(*pass trough*)
THIS^.pMqttPublishQueue := pMqttPublishQueue;
THIS^.MqttPublishTopicPrefix:=MQTTPublishPrefix;
THIS^.MQTTSubscribeTopicPrefix:=MQTTSubscribePrefix;
THIS^.pMqttPublishQueue:=pMqttPublishQueue;

// Dimmer specific
THIS^.OutputDimmer:=OutputDimmer;
THIS^.Qos_Dimm:=Qos_Dimm;
THIS^.Delta_Dimm:=Delta_Dimm;


SUPER^.InitBaseMqtt();
pMqttCallbackCollector^.put(instance:= THIS^); // register the FB agains the collector so mqtt events can be received
END_METHOD

METHOD InitMqttDiscovery
VAR_INPUT
	Device: POINTER TO FB_PLC_MQTT_DISCOVERY_DEVICE;
	Name: STRING(255);
	overruleId: STRING(255) := '';
	meta: STRING(255) := '';
END_VAR
VAR
	id: STRING(255);
END_VAR
IF InitMqttDone AND NOT initMqttDiscoveryDone THEN
	
	IF CommonTypesAndFunctions.StrEquals(str1:= ADR(overruleId), str2:= ADR('')) THEN
		id := CONCAT(CONCAT(THIS^.DeviceName,'_'), THIS^.InstanceNamePt^); // 'FB_DI_PB_003'
	ELSE
		id := overruleId; // 'MY_PH_GND_HALL_01'
	END_IF
	
	Device^.CreateLightDimmerEntity(
		Name := name,
		Id := Id,
		Meta := meta,
		CommandTopic := CONCAT(THIS^.MQTTSubscribeTopic,'/Q'),
		PayloadOn := 'TRUE',
		PayloadOff := 'FALSE',
		StateTopic := CONCAT(THIS^.MQTTPublishTopic,'/Q'),
		BrightnessCommandTopic := CONCAT(THIS^.MQTTSubscribeTopic,'/OUT'),
		BrightnessStateTopic := CONCAT(THIS^.MQTTPublishTopic,'/OUT'),
		BrightnessScale := 255,
		DmxChannel := THIS^.DmxChannel,
		DmxWidth := THIS^.DmxWidth,
		DmxUniverse := THIS^.DmxUniverse);

	initMqttDiscoveryDone := TRUE;
END_IF
END_METHOD

METHOD PublishReceived : BOOL
VAR_INPUT
	///Collection of recived Data
	Data: MQTT.CALLBACK_DATA;
END_VAR
//first check if Mqtt is initialized, otherwise do nothing
IF NOT(InitMqttDone) THEN
	//mark the interface call from the collector as done
	PublishReceived := TRUE;
//check if the packet is for this FB
ELSIF CONCAT(MQTTSubscribeTopic,'/Q') =  Data.TopicOut^ THEN
	IF CommonTypesAndFunctions.StrEquals(str1:= Data.PayloadString, str2:= ADR('TRUE')) THEN
		MqttHighRequest := TRUE;
	ELSIF CommonTypesAndFunctions.StrEquals(str1:= Data.PayloadString, str2:= ADR('FALSE')) THEN
		MqttLowRequest := TRUE;
	END_IF;
	
ELSIF CONCAT(MQTTSubscribeTopic,'/OUT') =  Data.TopicOut^ THEN
	IF OSCAT_BASIC.IS_CC(str:= Data.PayloadString^,cmp:='0123456789.') AND THIS^.PRIO_HIGH = FALSE THEN
		THIS^.OUT_Target:=STRING_TO_BYTE(Data.PayloadString^);
		THIS^.SoftDimToValue:=TRUE;
	END_IF
	
	
// Legacy! backwards compatiably with /+ topics instead of /#
ELSIF CommonTypesAndFunctions.StrEqualsAtStart(str1:= ADR(MQTTSubscribeTopic), str2:= Data.TopicOut) THEN
	//mark the interface call from the collector as done
	PublishReceived := TRUE;
	//now process the data
	IF CommonTypesAndFunctions.StrEquals(str1:= Data.PayloadString, str2:= ADR('TRUE')) THEN
		MqttHighRequest := TRUE;
	ELSIF CommonTypesAndFunctions.StrEquals(str1:= Data.PayloadString, str2:= ADR('FALSE')) THEN
		MqttLowRequest := TRUE;
	ELSIF OSCAT_BASIC.IS_CC(str:= Data.PayloadString^,cmp:='0123456789.') AND THIS^.PRIO_HIGH = FALSE THEN
		THIS^.OUT_Target:=STRING_TO_BYTE(Data.PayloadString^);
		THIS^.SoftDimToValue:=TRUE;
	END_IF
END_IF
END_METHOD

END_FUNCTION_BLOCK

// FB_VIRTUAL_INT_MQTT
{attribute 'reflection' := ''}
FUNCTION_BLOCK FB_VIRTUAL_INT_MQTT EXTENDS FB_MQTT_BASE IMPLEMENTS MQTT.MQTT_SUBSCRIBE_CALLBACK
VAR_INPUT
	IN: INT;
END_VAR
VAR_OUTPUT
	OUT: INT;
END_VAR
VAR
	/// Refelection: object's full instance name
	{attribute 'instance-path' := ''}
	{attribute 'noinit'}
	InstancePath: STRING;
	Startup: BOOL := TRUE;
	UpdateFlag: BOOL;
	VirtualMode: VIRTUAL_MODES;
	DefaultValue: INT;
	SetDefaultValueStartup: BOOL;
	PublishAtStartup: BOOL;
	UsePersistentAtStartup: BOOL;
	ConfirmReceival: BOOL;
	MqttMessageReceived: BOOL;
	PreviousIn: INT;
END_VAR
VAR PERSISTENT
	/// To retain output state through powercycles
	PreviousState: INT;
END_VAR

IF VirtualMode = VIRTUAL_MODES.Output THEN
	IF (Startup AND PublishAtStartup) OR (UpdateFlag OR IN <> PreviousIn) AND InitMqttDone THEN
	pMqttPublishQueue^.AddMessage(
		Payload := INT_TO_STRING(IN),
		Topic := CONCAT(MqttPublishTopicPrefix^, MqttPublishTopicSuffix),
		Qos := MqttQos,
		MqttRetain := MqttRetain
	);
	Startup:=FALSE;
	UpdateFlag := FALSE;
	PreviousIn := IN;
	END_IF
ELSIF VirtualMode = VIRTUAL_MODES.Input THEN
	IF Startup AND SetDefaultValueStartup THEN
		OUT := DefaultValue;
	ELSIF UsePersistentAtStartup THEN
		OUT := PreviousState;
	END_IF	
	
	IF ((Startup AND PublishAtStartup) OR (ConfirmReceival AND MqttMessageReceived)) AND InitMqttDone THEN
	pMqttPublishQueue^.AddMessage(
		Payload := INT_TO_STRING(OUT),
		Topic := CONCAT(MqttPublishTopicPrefix^, MqttPublishTopicSuffix),
		Qos := MqttQos,
		MqttRetain := MqttRetain
	);
	Startup:=FALSE;
	MqttMessageReceived := FALSE;
	PreviousState:=OUT;
	END_IF		
	
END_IF

METHOD ConfigureFunctionBlockAsVirtualInput : BOOL
VAR_INPUT
	DefaultValue: INT;
	SetDefaultValueStartup: BOOL;
	PublishAtStartup: BOOL;
	UsePersistentAtStartup: BOOL;
	ConfirmReceival: BOOL;
END_VAR
THIS^.DefaultValue:=DefaultValue;
THIS^.SetDefaultValueStartup:=SetDefaultValueStartup;
THIS^.PublishAtStartup:=PublishAtStartup;
THIS^.UsePersistentAtStartup:=UsePersistentAtStartup;
THIS^.ConfirmReceival:=ConfirmReceival;
THIS^.VirtualMode:=VIRTUAL_MODES.Input;
END_METHOD

METHOD ConfigureFunctionBlockAsVirtualOutput : BOOL
VAR_INPUT
	PublishAtStartup: BOOL;
END_VAR
THIS^.PublishAtStartup:=PublishAtStartup;
THIS^.VirtualMode:=VIRTUAL_MODES.Output;
END_METHOD

METHOD InitMqtt
VAR_INPUT
	MQTTPublishPrefix: POINTER TO STRING;
	MQTTSubscribePrefix: POINTER TO STRING;
	pMqttPublishQueue: POINTER TO FB_MqttPublishQueue;
	pMqttCallbackCollector: POINTER TO MQTT.CallbackCollector;
	MqttQos: MQTT.QoS;
	MqttRetain: BOOL;
END_VAR
InitMqttDone := TRUE;

SUPER^._InstancePath := THIS^.InstancePath; // Due to reflection its location is important

(*pass trough*)
THIS^.pMqttPublishQueue := pMqttPublishQueue;
THIS^.MqttPublishTopicPrefix:=MQTTPublishPrefix;
THIS^.MQTTSubscribeTopicPrefix:=MQTTSubscribePrefix;
THIS^.pMqttPublishQueue:=pMqttPublishQueue;
THIS^.MqttQos:=MqttQos;
THIS^.MqttRetain:=MqttRetain;


SUPER^.InitBaseMqtt();
pMqttCallbackCollector^.put(instance:= THIS^); // register the FB agains the collector so mqtt events can be received
END_METHOD

METHOD PublishReceived : BOOL
VAR_INPUT
	///Collection of recived Data
	Data: MQTT.CALLBACK_DATA;
END_VAR
//first check if Mqtt is initialized and FB in input mode, otherwise do nothing
IF NOT(InitMqttDone) AND VirtualMode <> VIRTUAL_MODES.Input THEN
	//mark the interface call from the collector as done
	PublishReceived := TRUE;
//check if the packet is for this FB
ELSIF CommonTypesAndFunctions.StrEquals(str1:= ADR(MQTTSubscribeTopic), str2:= Data.TopicOut) THEN
	//mark the interface call from the collector as done
	PublishReceived := TRUE;
	//process the data
	IF OSCAT_BASIC.IS_NUM(str:= Data.PayloadString^) THEN
		THIS^.OUT := STRING_TO_INT(Data.PayloadString^);	
		MqttMessageReceived := TRUE;	
	END_IF
END_IF
END_METHOD

METHOD SetValue : BOOL
VAR_INPUT
	Value: INT;
END_VAR
THIS^.OUT:=Value;
THIS^.UpdateFlag:=TRUE;
END_METHOD

END_FUNCTION_BLOCK

// FB_VIRTUAL_BOOL_MQTT
{attribute 'reflection' := ''}
FUNCTION_BLOCK FB_VIRTUAL_BOOL_MQTT EXTENDS FB_MQTT_BASE IMPLEMENTS MQTT.MQTT_SUBSCRIBE_CALLBACK
VAR_INPUT
	IN: BOOL;
END_VAR
VAR_OUTPUT
	OUT: BOOL;
END_VAR
VAR
	/// Refelection: object's full instance name
	{attribute 'instance-path' := ''}
	{attribute 'noinit'}
	InstancePath: STRING;
	Startup: BOOL := TRUE;
	UpdateFlag: BOOL;
	VirtualMode: VIRTUAL_MODES;
	DefaultValue: BOOL;
	SetDefaultValueStartup: BOOL;
	PublishAtStartup: BOOL;
	UsePersistentAtStartup: BOOL;
	ConfirmReceival: BOOL;
	MqttMessageReceived: BOOL;
	PreviousIn: BOOL;
END_VAR
VAR PERSISTENT
	/// To retain output state through powercycles
	PreviousState: BOOL;
END_VAR

IF VirtualMode = VIRTUAL_MODES.Output THEN
	IF (Startup AND PublishAtStartup) OR (UpdateFlag OR IN <> PreviousIn) AND InitMqttDone THEN
	pMqttPublishQueue^.AddMessage(
		Payload := BOOL_TO_STRING(IN),
		Topic := CONCAT(MqttPublishTopicPrefix^, MqttPublishTopicSuffix),
		Qos := MqttQos,
		MqttRetain := MqttRetain
	);
	Startup:=FALSE;
	UpdateFlag := FALSE;
	PreviousIn := IN;
	END_IF
ELSIF VirtualMode = VIRTUAL_MODES.Input THEN
	IF Startup AND SetDefaultValueStartup THEN
		OUT := DefaultValue;
	ELSIF UsePersistentAtStartup THEN
		OUT := PreviousState;
	END_IF	
	
	IF ((Startup AND PublishAtStartup) OR (ConfirmReceival AND MqttMessageReceived)) AND InitMqttDone THEN
	pMqttPublishQueue^.AddMessage(
		Payload := BOOL_TO_STRING(OUT),
		Topic := CONCAT(MqttPublishTopicPrefix^, MqttPublishTopicSuffix),
		Qos := MqttQos,
		MqttRetain := MqttRetain
	);
	Startup:=FALSE;
	MqttMessageReceived := FALSE;
	PreviousState:=OUT;
	END_IF		
	
END_IF

METHOD ConfigureFunctionBlockAsVirtualInput : BOOL
VAR_INPUT
	DefaultValue: BOOL;
	SetDefaultValueStartup: BOOL;
	PublishAtStartup: BOOL;
	UsePersistentAtStartup: BOOL;
	ConfirmReceival: BOOL;
END_VAR
THIS^.DefaultValue:=DefaultValue;
THIS^.SetDefaultValueStartup:=SetDefaultValueStartup;
THIS^.PublishAtStartup:=PublishAtStartup;
THIS^.UsePersistentAtStartup:=UsePersistentAtStartup;
THIS^.ConfirmReceival:=ConfirmReceival;
THIS^.VirtualMode:=VIRTUAL_MODES.Input;
END_METHOD

METHOD ConfigureFunctionBlockAsVirtualOutput : BOOL
VAR_INPUT
	PublishAtStartup: BOOL;
END_VAR
THIS^.PublishAtStartup:=PublishAtStartup;
THIS^.VirtualMode:=VIRTUAL_MODES.Output;
END_METHOD

METHOD InitMqtt
VAR_INPUT
	MQTTPublishPrefix: POINTER TO STRING;
	MQTTSubscribePrefix: POINTER TO STRING;
	pMqttPublishQueue: POINTER TO FB_MqttPublishQueue;
	pMqttCallbackCollector: POINTER TO MQTT.CallbackCollector;
	MqttQos: MQTT.QoS;
	MqttRetain: BOOL;
END_VAR
InitMqttDone := TRUE;

SUPER^._InstancePath := THIS^.InstancePath; // Due to reflection its location is important

(*pass trough*)
THIS^.pMqttPublishQueue := pMqttPublishQueue;
THIS^.MqttPublishTopicPrefix:=MQTTPublishPrefix;
THIS^.MQTTSubscribeTopicPrefix:=MQTTSubscribePrefix;
THIS^.pMqttPublishQueue:=pMqttPublishQueue;
THIS^.MqttQos:=MqttQos;
THIS^.MqttRetain:=MqttRetain;


SUPER^.InitBaseMqtt();
pMqttCallbackCollector^.put(instance:= THIS^); // register the FB agains the collector so mqtt events can be received
END_METHOD

METHOD PublishReceived : BOOL
VAR_INPUT
	///Collection of recived Data
	Data: MQTT.CALLBACK_DATA;
END_VAR
//first check if Mqtt is initialized and FB in input mode, otherwise do nothing
IF NOT(InitMqttDone) AND VirtualMode <> VIRTUAL_MODES.Input THEN
	//mark the interface call from the collector as done
	PublishReceived := TRUE;
//check if the packet is for this FB
ELSIF CommonTypesAndFunctions.StrEquals(str1:= ADR(MQTTSubscribeTopic), str2:= Data.TopicOut) THEN
	//mark the interface call from the collector as done
	PublishReceived := TRUE;
	//process the data
	IF CommonTypesAndFunctions.StrEquals(str1:= Data.PayloadString, str2:= ADR('TRUE')) THEN
		THIS^.OUT := TRUE;
		MqttMessageReceived := TRUE;
	END_IF
	IF CommonTypesAndFunctions.StrEquals(str1:= Data.PayloadString, str2:= ADR('FALSE')) THEN
		THIS^.OUT := FALSE;
		MqttMessageReceived := TRUE;
	END_IF
END_IF
END_METHOD

METHOD SetValue : BOOL
VAR_INPUT
	Value: BOOL;
END_VAR
THIS^.OUT:=Value;
THIS^.UpdateFlag:=TRUE;
END_METHOD

END_FUNCTION_BLOCK

// FB_VIRTUAL_STRING_MQTT
{attribute 'reflection' := ''}
FUNCTION_BLOCK FB_VIRTUAL_STRING_MQTT EXTENDS FB_MQTT_BASE IMPLEMENTS MQTT.MQTT_SUBSCRIBE_CALLBACK
VAR_INPUT
	IN: STRING;
END_VAR
VAR_OUTPUT
	OUT: STRING;
END_VAR
VAR
	/// Refelection: object's full instance name
	{attribute 'noinit'}
	{attribute 'instance-path' := ''}
	InstancePath: STRING;
	Startup: BOOL := TRUE;
	UpdateFlag: BOOL;
	VirtualMode: VIRTUAL_MODES;
	DefaultValue: STRING;
	SetDefaultValueStartup: BOOL;
	PublishAtStartup: BOOL;
	UsePersistentAtStartup: BOOL;
	ConfirmReceival: BOOL;
	MqttMessageReceived: BOOL;
	PreviousIn: STRING;
END_VAR
VAR PERSISTENT
	/// To retain output state through powercycles
	PreviousState: STRING;
END_VAR

IF VirtualMode = VIRTUAL_MODES.Output THEN
	IF (Startup AND PublishAtStartup) OR (UpdateFlag OR IN <> PreviousIn) AND InitMqttDone THEN
	pMqttPublishQueue^.AddMessage(
		Payload := IN,
		Topic := CONCAT(MqttPublishTopicPrefix^, MqttPublishTopicSuffix),
		Qos := MqttQos,
		MqttRetain := MqttRetain
	);
	Startup:=FALSE;
	UpdateFlag := FALSE;
	PreviousIn := IN;
	END_IF
ELSIF VirtualMode = VIRTUAL_MODES.Input THEN
	IF Startup AND SetDefaultValueStartup THEN
		OUT := DefaultValue;
	ELSIF UsePersistentAtStartup THEN
		OUT := PreviousState;
	END_IF	
	
	IF ((Startup AND PublishAtStartup) OR (ConfirmReceival AND MqttMessageReceived)) AND InitMqttDone THEN
	pMqttPublishQueue^.AddMessage(
		Payload := OUT,
		Topic := CONCAT(MqttPublishTopicPrefix^, MqttPublishTopicSuffix),
		Qos := MqttQos,
		MqttRetain := MqttRetain
	);
	Startup:=FALSE;
	MqttMessageReceived := FALSE;
	PreviousState:=OUT;
	END_IF		
	
END_IF

METHOD ConfigureFunctionBlockAsVirtualInput : BOOL
VAR_INPUT
	DefaultValue: STRING;
	SetDefaultValueStartup: BOOL;
	PublishAtStartup: BOOL;
	UsePersistentAtStartup: BOOL;
	ConfirmReceival: BOOL;
END_VAR
THIS^.DefaultValue:=DefaultValue;
THIS^.SetDefaultValueStartup:=SetDefaultValueStartup;
THIS^.PublishAtStartup:=PublishAtStartup;
THIS^.UsePersistentAtStartup:=UsePersistentAtStartup;
THIS^.ConfirmReceival:=ConfirmReceival;
THIS^.VirtualMode:=VIRTUAL_MODES.Input;
END_METHOD

METHOD ConfigureFunctionBlockAsVirtualOutput : BOOL
VAR_INPUT
	PublishAtStartup: BOOL;
END_VAR
THIS^.PublishAtStartup:=PublishAtStartup;
THIS^.VirtualMode:=VIRTUAL_MODES.Output;
END_METHOD

METHOD InitMqtt
VAR_INPUT
	MQTTPublishPrefix: POINTER TO STRING;
	MQTTSubscribePrefix: POINTER TO STRING;
	pMqttPublishQueue: POINTER TO FB_MqttPublishQueue;
	pMqttCallbackCollector: POINTER TO MQTT.CallbackCollector;
	MqttQos: MQTT.QoS;
	MqttRetain: BOOL;
END_VAR
InitMqttDone := TRUE;

SUPER^._InstancePath := THIS^.InstancePath; // Due to reflection its location is important

(*pass trough*)
THIS^.pMqttPublishQueue := pMqttPublishQueue;
THIS^.MqttPublishTopicPrefix:=MQTTPublishPrefix;
THIS^.MQTTSubscribeTopicPrefix:=MQTTSubscribePrefix;
THIS^.pMqttPublishQueue:=pMqttPublishQueue;
THIS^.MqttQos:=MqttQos;
THIS^.MqttRetain:=MqttRetain;


SUPER^.InitBaseMqtt();
pMqttCallbackCollector^.put(instance:= THIS^); // register the FB agains the collector so mqtt events can be received
END_METHOD

METHOD PublishReceived : BOOL
VAR_INPUT
	///Collection of recived Data
	Data: MQTT.CALLBACK_DATA;
END_VAR
//first check if Mqtt is initialized and FB in input mode, otherwise do nothing
IF NOT(InitMqttDone) AND VirtualMode <> VIRTUAL_MODES.Input THEN
	//mark the interface call from the collector as done
	PublishReceived := TRUE;
//check if the packet is for this FB
ELSIF CommonTypesAndFunctions.StrEquals(str1:= ADR(MQTTSubscribeTopic), str2:= Data.TopicOut) THEN
	//mark the interface call from the collector as done
	PublishReceived := TRUE;
	//process the data
	THIS^.OUT := Data.PayloadString^;	
	MqttMessageReceived := TRUE;
END_IF
END_METHOD

METHOD SetValue : BOOL
VAR_INPUT
	Value: STRING;
END_VAR
THIS^.OUT:=Value;
THIS^.UpdateFlag:=TRUE;
END_METHOD

END_FUNCTION_BLOCK

// FB_VIRTUAL_REAL_MQTT
{attribute 'reflection' := ''}
FUNCTION_BLOCK FB_VIRTUAL_REAL_MQTT EXTENDS FB_MQTT_BASE IMPLEMENTS MQTT.MQTT_SUBSCRIBE_CALLBACK
VAR_INPUT
	IN: REAL;
END_VAR
VAR_OUTPUT
	OUT: REAL;
END_VAR
VAR
	/// Refelection: object's full instance name
	{attribute 'instance-path' := ''}
	{attribute 'noinit'}
	InstancePath: STRING;
	Startup: BOOL := TRUE;
	UpdateFlag: BOOL;
	VirtualMode: VIRTUAL_MODES;
	DefaultValue: REAL;
	SetDefaultValueStartup: BOOL;
	PublishAtStartup: BOOL;
	UsePersistentAtStartup: BOOL;
	ConfirmReceival: BOOL;
	MqttMessageReceived: BOOL;
	PreviousIn: REAL;
END_VAR
VAR PERSISTENT
	/// To retain output state through powercycles
	PreviousState: REAL;
END_VAR

IF VirtualMode = VIRTUAL_MODES.Output THEN
	IF (Startup AND PublishAtStartup) OR (UpdateFlag OR IN <> PreviousIn) AND InitMqttDone THEN
	pMqttPublishQueue^.AddMessage(
		Payload := REAL_TO_STRING(IN),
		Topic := CONCAT(MqttPublishTopicPrefix^, MqttPublishTopicSuffix),
		Qos := MqttQos,
		MqttRetain := MqttRetain
	);
	Startup:=FALSE;
	UpdateFlag := FALSE;
	PreviousIn := IN;
	END_IF
ELSIF VirtualMode = VIRTUAL_MODES.Input THEN
	IF Startup AND SetDefaultValueStartup THEN
		OUT := DefaultValue;
	ELSIF UsePersistentAtStartup THEN
		OUT := PreviousState;
	END_IF	
	
	IF ((Startup AND PublishAtStartup) OR (ConfirmReceival AND MqttMessageReceived)) AND InitMqttDone THEN
	pMqttPublishQueue^.AddMessage(
		Payload := REAL_TO_STRING(OUT),
		Topic := CONCAT(MqttPublishTopicPrefix^, MqttPublishTopicSuffix),
		Qos := MqttQos,
		MqttRetain := MqttRetain
	);
	Startup:=FALSE;
	MqttMessageReceived := FALSE;
	PreviousState:=OUT;
	END_IF		
	
END_IF

METHOD ConfigureFunctionBlockAsVirtualInput : BOOL
VAR_INPUT
	DefaultValue: REAL;
	SetDefaultValueStartup: BOOL;
	PublishAtStartup: BOOL;
	UsePersistentAtStartup: BOOL;
	ConfirmReceival: BOOL;
END_VAR
THIS^.DefaultValue:=DefaultValue;
THIS^.SetDefaultValueStartup:=SetDefaultValueStartup;
THIS^.PublishAtStartup:=PublishAtStartup;
THIS^.UsePersistentAtStartup:=UsePersistentAtStartup;
THIS^.ConfirmReceival:=ConfirmReceival;
THIS^.VirtualMode:=VIRTUAL_MODES.Input;
END_METHOD

METHOD ConfigureFunctionBlockAsVirtualOutput : BOOL
VAR_INPUT
	PublishAtStartup: BOOL;
END_VAR
THIS^.PublishAtStartup:=PublishAtStartup;
THIS^.VirtualMode:=VIRTUAL_MODES.Output;
END_METHOD

METHOD InitMqtt
VAR_INPUT
	MQTTPublishPrefix: POINTER TO STRING;
	MQTTSubscribePrefix: POINTER TO STRING;
	pMqttPublishQueue: POINTER TO FB_MqttPublishQueue;
	pMqttCallbackCollector: POINTER TO MQTT.CallbackCollector;
	MqttQos: MQTT.QoS;
	MqttRetain: BOOL;
END_VAR
InitMqttDone := TRUE;

SUPER^._InstancePath := THIS^.InstancePath; // Due to reflection its location is important

(*pass trough*)
THIS^.pMqttPublishQueue := pMqttPublishQueue;
THIS^.MqttPublishTopicPrefix:=MQTTPublishPrefix;
THIS^.MQTTSubscribeTopicPrefix:=MQTTSubscribePrefix;
THIS^.pMqttPublishQueue:=pMqttPublishQueue;
THIS^.MqttQos:=MqttQos;
THIS^.MqttRetain:=MqttRetain;


SUPER^.InitBaseMqtt();
pMqttCallbackCollector^.put(instance:= THIS^); // register the FB agains the collector so mqtt events can be received
END_METHOD

METHOD PublishReceived : BOOL
VAR_INPUT
	///Collection of recived Data
	Data: MQTT.CALLBACK_DATA;
END_VAR
//first check if Mqtt is initialized and FB in input mode, otherwise do nothing
IF NOT(InitMqttDone) AND VirtualMode <> VIRTUAL_MODES.Input THEN
	//mark the interface call from the collector as done
	PublishReceived := TRUE;
//check if the packet is for this FB
ELSIF CommonTypesAndFunctions.StrEquals(str1:= ADR(MQTTSubscribeTopic), str2:= Data.TopicOut) THEN
	//mark the interface call from the collector as done
	PublishReceived := TRUE;
	//process the data
	THIS^.OUT := STRING_TO_REAL(Data.PayloadString^);	
	MqttMessageReceived := TRUE;	
END_IF
END_METHOD

METHOD SetValue : BOOL
VAR_INPUT
	Value: REAL;
END_VAR
THIS^.OUT:=Value;
THIS^.UpdateFlag:=TRUE;
END_METHOD

END_FUNCTION_BLOCK

// HomeAutomation/PRG's/PLC_PRG_MQTT
PROGRAM PLC_PRG_MQTT
VAR
	MQTTClient				:MQTT.MQTTClient;
	MQTT_IN_OUT				:MQTT.MQTT_IN_OUT;
	MQTTInfo				:MQTT.MQTT_INFO;
	MQTTBirthMessage		:MQTT_MESSAGE;;
	MQTTBirthHartbeat		:OSCAT_BASIC.GEN_PULSE;
	MQTTConnectTrigger		:Standard.R_TRIG;
	MQTTPublishBirth		:BOOL:=TRUE;
	MQTTBirthPublisher		:FB_MqttPublishWorker;

	(* variables for MQTT setup *)
	initMqtt				:BOOL;
	icounter				:UDINT;
	
	(* variables for MQTT publishing *)
	ipublishers				:UDINT:=40;
	publishers				:ARRAY[0..39] OF FB_MqttPublishWorker;
	
	(* variables to work with Mqttbuffer *)
	i : UDINT;
	
	(* variables for MQTT subscribing *)
	subscriber_FB_OUTPUT_SWITCH_MQTT:MQTT.MQTTSubscribe;
	subscriber_FB_OUTPUT_COVER_MQTT:MQTT.MQTTSubscribe;	
	subscriber_FB_VIRTUAL_MQTT:MQTT.MQTTSubscribe;	
	subscriber_FB_DIMMER_MQTT:MQTT.MQTTSubscribe;
	subscriber_FB_RS485_MQTT:MQTT.MQTTSubscribe;	
END_VAR

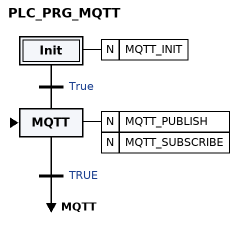
INITIAL_STEP Init:
    MQTT_INIT(N);
END_STEP
TRANSITION FROM Init TO MQTT
    := True;
END_TRANSITION
STEP MQTT:
    MQTT_PUBLISH(N);
    MQTT_SUBSCRIBE(N);
END_STEP
TRANSITION FROM MQTT TO MQTT
    := TRUE;
END_TRANSITION

ACTION MQTT_INIT:

IF NOT initMqtt THEN
	initMqtt := TRUE;
	(* Basic MQTT config *)
	MQTT_IN_OUT.ClientID := MqttVariables.clientID;
	
	(* Set the LWT topic / payload *)
	MQTT_IN_OUT.BuildWillTopicAndMessage := FALSE;
	MQTT_IN_OUT.WillTopicBase := '';
	MQTT_IN_OUT.ClientWillTopic := MqttVariables.MqttAvailabilityTopic;
	MQTT_IN_OUT.ClientWillMessage := MqttVariables.MqttAvailabilityOfflinePayload;
	
	(* Set the birth message *)
	MQTTBirthMessage.Payload := MqttVariables.MqttAvailabilityOnlinePayload;
	MQTTBirthMessage.Topic := MqttVariables.MqttAvailabilityTopic;
	MQTTBirthMessage.Qos := MqttVariables.MQTT_QOS_EXACTLY_ONCE;
	MQTTBirthMessage.MqttRetain := FALSE;
	
	(* Configure the rising edge detector to detect a connect/reconnect to the broker, used for  birth message *)
	MQTTConnectTrigger(CLK := MQTTInfo.MQTT_CONNECTED);
	
	(* Configure the dedicated MQTTBirth publisher *)
	MQTTBirthPublisher.Init(inputMQTT_IN_OUT:= ADR(MQTT_IN_OUT));
	
	(* Configure the pulse generator for the birth message hartbeat *)
	 MQTTBirthHartbeat(ENQ:=TRUE, PTH:=T#0S, PTL:=MqttVariables.MQTTAvailabilityHartbeatTime);
	
	(* INIT MQTT PUBLISH STUFF *)
	FOR icounter := 0 TO (ipublishers-1) DO		
		publishers[icounter].Init(inputMQTT_IN_OUT:= ADR(MQTT_IN_OUT));
	END_FOR 
	
	(* INIT MQTT SUBSCRIBE STUFF *)
	subscriber_FB_OUTPUT_SWITCH_MQTT.SetMqttInOut(MQTT_IN_OUT:= MQTT_IN_OUT);	
	subscriber_FB_OUTPUT_COVER_MQTT.SetMqttInOut(MQTT_IN_OUT:= MQTT_IN_OUT);
	subscriber_FB_VIRTUAL_MQTT.SetMqttInOut(MQTT_IN_OUT:= MQTT_IN_OUT);	
	subscriber_FB_DIMMER_MQTT.SetMqttInOut(MQTT_IN_OUT:= MQTT_IN_OUT);
	subscriber_FB_RS485_MQTT.SetMqttInOut(MQTT_IN_OUT:= MQTT_IN_OUT);
END_IF
END_ACTION

ACTION MQTT_PUBLISH:
(* set user led green if connected to MQTT broker, flashing red if not *)
(* é!COCKPIT version *)
(* LED_1_BrokerStatus(eID:=eLedID.AppLED_1, xOpen:=TRUE );
IF(MQTTClient.connected) THEN
	LED_1_BrokerStatus.SetStatic(eLedColor.Green);
ELSE
	LED_1_BrokerStatus.SetFlash(T#1S,eLedColor.Red, eLedColor.Off);  
END_IF *)
(* Codesys 3S version *)
(*
IF MQTTClient.connected THEN
     PFC.SetLed(which:=PFC.LED.U1, how:=PFC.LedState.STATIC_GRN);
ELSE
     PFC.SetLed(which:=PFC.LED.U1, how:=PFC.LedState.BLINK_RED);
END_IF 
*)

(* allow the rising edge detector to detect a connect/reconnect to the broker, used for  birth message *)
MQTTConnectTrigger(CLK := MQTTInfo.MQTT_CONNECTED);

(* allow the pulse generator to generate a pulse, used for birth message hartbeat *)
MQTTBirthHartbeat(ENQ:=TRUE, PTH:=T#0S, PTL:=MqttVariables.MQTTAvailabilityHartbeatTime);

(* Check if this is a new connection due to startup or connection issues *)
IF initMqtt AND (MQTTConnectTrigger.Q OR MQTTBirthHartbeat.Q) THEN
	MQTTPublishBirth := TRUE;
END_IF

(* On connect or reconnect publish a birth message using the dedicated birth publisher *)
IF MQTTPublishBirth THEN
	MQTTBirthPublisher.PublishMessage(MqttMessage := MQTTBirthMessage);
	MQTTPublishBirth:=FALSE;
END_IF


(* Check if Mqtt is initialized AND if there are elements on the queue to process AND if a MQTTbirthmessage has been published successfully *)
IF initMqtt AND NOT(MqttVariables.fbMqttPublishQueue.EMPTY) AND MQTTPublishBirth = FALSE AND MQTTBirthPublisher.SendDone THEN	
	(* Loop through all free publishers untill there are no more elements in the queue or no more free publishers *)
	FOR i:=0 TO (ipublishers-1) DO			
		(* use the publishers that are free  *)
		IF publishers[i].SendDone AND NOT(MqttVariables.fbMqttPublishQueue.EMPTY) THEN	
			(* Pass message from the queue to a publisher *)
			publishers[i].PublishMessage(MqttMessage:= MqttVariables.fbMqttPublishQueue.GetMessage());
		ELSIF MqttVariables.fbMqttPublishQueue.EMPTY THEN
			(* Queue is empty, jump out of the for loop	*)
			EXIT;	
		END_IF
	END_FOR
END_IF


(* If MQTT is initialized, let the MqttPublishWorkers do their work *)
IF initMqtt THEN	
	MQTT_IN_OUT.clientFB(
		MQTT_IN_OUT:= MQTT_IN_OUT, 
		ENABLE:= TRUE, 
		URL:= MQttVariables.broker, 
		TIMEOUT:= T#1S, 
		TLS:= FALSE);		
		
	MQTTBirthPublisher();
	
	FOR i := 0 TO (ipublishers-1) DO
  		publishers[i]();
	END_FOR

END_IF
END_ACTION

ACTION MQTT_SUBSCRIBE:
(* If MQTT is initialized, let the subscriber(s) do its work *)
IF initMqtt THEN
	
	MQTT_IN_OUT.clientFB(
		MQTT_IN_OUT:= MQTT_IN_OUT, 
		ENABLE:= TRUE, 
		URL:= MqttVariables.broker, 
		TIMEOUT:= T#1S, 
		TLS:= FALSE);

	subscriber_FB_OUTPUT_SWITCH_MQTT(
		Subscribe:= TRUE, 
		Topic:= ADR(MqttVariables.MqttSubSwitchTopic), 
		QoSSubscribe:= MqttVariables.MQTT_QOS_EXACTLY_ONCE, 
		ExpectingString:= TRUE, 
		Callback:= MqttVariables.collector_FB_OUTPUT_SWITCH_MQTT,
	);	
	subscriber_FB_OUTPUT_COVER_MQTT(
		Subscribe:= TRUE, 
		Topic:= ADR(MqttVariables.MqttSubCoverTopic), 
		QoSSubscribe:= MqttVariables.MQTT_QOS_EXACTLY_ONCE, 
		ExpectingString:= TRUE, 
		Callback:= MqttVariables.collector_FB_OUTPUT_COVER_MQTT,
	);	
	subscriber_FB_VIRTUAL_MQTT(
		Subscribe:= TRUE, 
		Topic:= ADR(MqttVariables.MqttSubVirtualTopic), 
		QoSSubscribe:= MqttVariables.MQTT_QOS_EXACTLY_ONCE, 
		ExpectingString:= TRUE, 
		Callback:= MqttVariables.collector_FB_VIRTUAL_MQTT,
	);
	subscriber_FB_DIMMER_MQTT(
		Subscribe:= TRUE, 
		Topic:= ADR(MqttVariables.MqttSubDimmerTopic), 
		QoSSubscribe:= MqttVariables.MQTT_QOS_EXACTLY_ONCE, 
		ExpectingString:= TRUE, 
		Callback:= MqttVariables.collector_FB_DIMMER_MQTT,
	);
	subscriber_FB_RS485_MQTT(
		Subscribe:= TRUE, 
		Topic:= ADR(MqttVariables.MqttSubRS485Topic), 
		QoSSubscribe:= MqttVariables.MQTT_QOS_EXACTLY_ONCE,
		ExpectingString:= TRUE, 
		Callback:= MqttVariables.collector_FB_RS485_MQTT,
	);
END_IF
END_ACTION

END_PROGRAM

// Mqtt/FB_MqttPublishWorker
FUNCTION_BLOCK FB_MqttPublishWorker
VAR_OUTPUT
	SendDone: BOOL;
END_VAR
VAR
	LocalMqttMessage: MQTT_MESSAGE;
	InitDone: BOOL;
	RequestToSend: BOOL;
	Send: BOOL;
	publish: MQTT.MQTTPublish;
END_VAR

//need to call publish here because of FB nums
publish(
	Topic:= ADR(LocalMqttMessage.Topic), 
	PayloadString:= ADR(LocalMqttMessage.Payload), 
	PublishAsString:= TRUE, 
	QoSIn:= LocalMqttMessage.Qos, 
	MRetain:= LocalMqttMessage.MqttRetain, 
	send:= Send);
	
IF NOT InitDone THEN RETURN; END_IF

IF RequestToSend THEN
	Send := TRUE;
	SendDone := FALSE;
END_IF

IF publish.done THEN
	 SendDone := TRUE;
	 RequestToSend:=FALSE;
	 Send:=FALSE;
END_IF

METHOD Init
VAR_INPUT
	///Pointer MQTTT exchange strucure
	inputMQTT_IN_OUT: POINTER TO MQTT.MQTT_IN_OUT;
END_VAR
publish.SetMqttInOut(MQTT_IN_OUT := inputMQTT_IN_OUT^);

InitDone := TRUE;
SendDone := TRUE;
END_METHOD

METHOD PublishMessage
VAR_INPUT
	MqttMessage: MQTT_MESSAGE;
END_VAR
LocalMqttMessage := MqttMessage;

RequestToSend:=TRUE;
END_METHOD

END_FUNCTION_BLOCK

// HomeAutomation/PRG's/DMX_SEND
PROGRAM DMX_SEND
VAR
	Universe	: INT     :=1;
	IP_CONTROL2	: oscat_network.IP_CONTROL2;
	IP_C		: oscat_network.IP_C;
	S_BUF1		: oscat_network.NETWORK_BUFFER_SHORT;
	R_BUF1		: oscat_network.NETWORK_BUFFER_SHORT;
	error_send	: BOOL:= FALSE;
	i			: INT;
	init		: BOOL;
	start		: INT;
	size		: INT;
	LED_1_BrokerStatus		:FbAppLED;
	Step: INT:=0;
END_VAR

IF init = FALSE THEN
	init := TRUE;
	//https://art-net.org.uk/how-it-works/streaming-packets/artdmx-packet-definition/
	(* Write DMX header character in the buffer *) 
	S_BUF1.BUFFER [0]:= BYTE#16#41; // A
	S_BUF1.BUFFER [1]:= BYTE#16#72; // R	
	S_BUF1.BUFFER [2]:= BYTE#16#74; // T
	S_BUF1.BUFFER [3]:= BYTE#16#2D; // -
	S_BUF1.BUFFER [4]:= BYTE#16#4E; // N
	S_BUF1.BUFFER [5]:= BYTE#16#65; // E
	S_BUF1.BUFFER [6]:= BYTE#16#74; // T
	S_BUF1.BUFFER [7]:= BYTE#16#00; // 0 zero
	
	S_BUF1.BUFFER [8]:= BYTE#16#00;	// Opcode ArtDMX (0x5000) little endian
	S_BUF1.BUFFER [9]:= BYTE#16#50; // Opcode ArtDMX (0x5000) little endian
	
	S_BUF1.BUFFER [10]:= BYTE#16#00; // Protocol Version Hi (0)
	S_BUF1.BUFFER [11]:= BYTE#16#0E; // Protocol Version Lo (14)
	
	S_BUF1.BUFFER [12]:= BYTE#16#00; // Sequence
	S_BUF1.BUFFER [13]:= BYTE#16#00; // Physical
	
	S_BUF1.BUFFER [16]:= BYTE#16#02; // Length Hi
	S_BUF1.BUFFER [17]:= BYTE#16#00; // Length Lo (2 to 512, even)
	(* the DMX channels that are next have already been written to the buffer *) 
	
	IF Universe = 1 THEN
		S_BUF1.BUFFER [14]:= BYTE#16#01; // Universe little endian
		S_BUF1.BUFFER [15]:= BYTE#16#00; // Universe little endian
	END_IF
	IF Universe = 2 THEN
		S_BUF1.BUFFER [14]:= BYTE#16#02; // Universe little endian
		S_BUF1.BUFFER [15]:= BYTE#16#00; // Universe little endian
	END_IF
END_IF;


size := 512+18;
FOR i:= 0 TO size DO (* check whether the DMX values ​​in the global variable have changed *)
	// i+2 is strange, buffers are not the same, its often offset with 2 sometimes by 1, todo
	IF S_BUF1.BUFFER[i+18] <> DMXVariables.DMX.BUFFER[i+2] THEN
   		S_BUF1.BUFFER[i+18]:= DMXVariables.DMX.BUFFER[i+2];
		Step := 1;
	END_IF
END_FOR

S_BUF1.BUFFER [17]:= S_BUF1.BUFFER [17]; // low...
DMXVariables.DMX.BUFFER[0] := DMXVariables.DMX.BUFFER[0];
S_BUF1.BUFFER [18]:= S_BUF1.BUFFER [18];
DMXVariables.DMX.BUFFER[1] := DMXVariables.DMX.BUFFER[1];
S_BUF1.BUFFER [19]:= S_BUF1.BUFFER [19];
DMXVariables.DMX.BUFFER[2] := DMXVariables.DMX.BUFFER[2];
S_BUF1.BUFFER [20]:= S_BUF1.BUFFER [20];
DMXVariables.DMX.BUFFER[3] := DMXVariables.DMX.BUFFER[3];


CASE Step OF
	0:
		//passive
	
	1:
		IP_C.C_MODE := 1; (* Mode: UDP+ACTIVE+Port+IP *)
		IP_C.C_ENABLE := TRUE; (* Release connection *)
		IP_C.TIME_RESET := TRUE; (*Reset TIME monitoring * *)
		IP_C.R_OBSERVE := TRUE; (* Monitor data receive *)
		R_BUF1.SIZE:= 0; (* Reset Home length *)
		IP_C.C_IP:= oscat_network.IP4_DECODE (DMXVariables.IP);
		IP_C.C_PORT:= WORD#6454;
		
		S_BUF1.SIZE := size;
		Step:=2;
		
	2:
		IP_CONTROL2 (TIME_OUT:= T#1S, IP_C:= IP_C, S_BUF:= S_BUF1, R_BUF:= R_BUF1);
		
		IF IP_C.ERROR <> 0  THEN
			Step:=666;
		END_IF
	666:
		LED_1_BrokerStatus(eID:=eLedID.AppLED_1, xOpen:=TRUE );
		LED_1_BrokerStatus.SetFlash(T#2S,eLedColor.Red, eLedColor.Off);
		IF IP_C.ERROR = 33554432  THEN
		MqttVariables.PLC_Device.SendLogMessage(CONCAT('ERROR|DMX has a connection error ', DWORD_TO_STRING(IP_C.ERROR)));
		
		END_IF;
		
		error_send := TRUE;
		R_BUF1.SIZE := 0;
		IP_C.C_ENABLE:= FALSE; (* Enable connection establishment *) 
		IP_C.TIME_RESET:= FALSE;
		init:=FALSE;
	ELSE
	  Step := 0;
END_CASE



// Check IP_C1.error
// 33554432 = 0x02000000
// Initialization of the socket interface failed (only WinNT).
// code = 0x 02 00 00 00 (hexadecimal)
//           !   !    ! 
//           !   !    Receive error 
//           !   Send error
//           Connect error

END_PROGRAM

// HomeAutomation/PRG's/PRG_PING_DMX
PROGRAM PRG_PING_DMX
VAR
	PingTime: UDINT;
	DMXnodeReachable: UDINT;
	LED_1_BrokerStatus: FbAppLED;
END_VAR

(* Ping the DMX artNet node *)
DMXnodeReachable := SysSockPing(szIPAddress:=DMXVariables.IP, ulTimeout:=500, pulReplyTime:= ADR(PingTime));

IF DMXnodeReachable = 0 THEN
	LED_1_BrokerStatus.SetStatic(eLedColor.Green);
// 	MqttVariables.MQTT_logger.send('DMX ping OK');
ELSIF DMXnodeReachable = 5 THEN
	LED_1_BrokerStatus.SetFlash(T#1S,eLedColor.Red, eLedColor.Off);
	MqttVariables.PLC_Device.SendLogMessage('DMX ping Error');
END_IF

END_PROGRAM

// HomeAutomation/PRG's/PLC_PRG_RS485
PROGRAM PLC_PRG_RS485
VAR
	(* CODESYS 3S Version version*)
	(*
	xComPortOpen         : BOOL;
    xComPortError        : BOOL;
    rtsResult            : RTS_IEC_RESULT;	
    stComPortSettings    : SysCom.SysComSettings :=(
											ulBaudrate :=9600,
											byParity := 0,
											byStopBits:=1,
											ulTimeout :=500,
											ulBufferSize :=256,
											
											sPort:=SYS_COM_PORTS.SYS_COMPORT1											
										);
    hComPort             : RTS_IEC_HANDLE; 
    awReadBuffer         : ARRAY[0..124] OF WORD;        
    awWriteBuffer        : ARRAY[0..124] OF WORD;     
    fbModbusRequest      : IoDrvModbus.ModbusRequest2;
    eComError            : IoDrvModbus.MB_ErrorCodes;	
	*)
	
	(* é!COCKPIT version*)
	ModbusMaster  		: WagoAppPlcModbus.FbMbMasterSerial := (
											xConnect    := TRUE,
                                            udiBaudrate := 9600,
                                            usiDataBits := 8,
                                            eParity     := WagoTypesCom.eTTYParity.None,
                                            eStopBits   := WagoTypesCom.eTTYStopBits.One,
                                            eHandshake  := WagoTypesCom.eTTYHandshake.None,
                                            ePhysical   := WagoTypesCom.eTTYPhysicalLayer.RS485_HalfDuplex,
                                            eFrameType  := eMbFrameType.RTU,
                                            tTimeOut    := T#500MS
                                          );
	RtuQuery			: WagoAppPlcModbus.typMbQuery;
	RtuResponse			: WagoAppPlcModbus.typMbResponse;
	
	
	(* Shared variables for é!COCKPIT and CODESYS 3S Version *)
	Trigger				: BOOL:=FALSE;
	InitRS485			: BOOL:=FALSE;
	ActiveRtuQuery		: RS485_RtuQuery;
	RS485BusController 	: FB_RS485_BUSCONTROLLER;	
	

	(* RS485 *)
	FB_RS485_EASTRON_SDM220_1				: FB_RS485_EASTRON_SDM220_MQTT;
	FB_RS485_ESERA_1WIRE_GATEWAY_MQTT_HOME	: FB_RS485_ESERA_1WIRE_GATEWAY_MQTT;
	FB_RS485_DUCO_DUCOBOX_HOME				: FB_RS485_DUCO_DUCOBOX_MQTT;
END_VAR

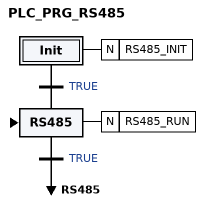
INITIAL_STEP Init:
    RS485_INIT(N);
END_STEP
TRANSITION FROM Init TO RS485
    := TRUE;
END_TRANSITION
STEP RS485:
    RS485_RUN(N);
END_STEP
TRANSITION FROM RS485 TO RS485
    := TRUE;
END_TRANSITION

ACTION RS485_INIT:
IF NOT InitRS485 THEN
	InitRS485 := TRUE;

(* INIT RS485 BUS CONTROLLER; CODESYS 3S Version version *)
(*
RS485BusController.Init(
	StartupDelay := T#5S,				(* Time to wait after startup to start using the bus, prevents boot delay issues when RS485 are not ready yet on startup *)		
	SilenceTime := T#50MS,				(* Silence time between two requests, important to not get faulty data on bus *)
	BusTrigger := ADR(Trigger),			(* Pointer to the bool used to initiate bus requests *)
	BusData := ADR(awReadBuffer),		(* Pointer to the array containing the bus response data *)
	BusError := ADR(xComPortError)		(* Pointer to the bus error bool *)
);
*)

(* INIT RS485 BUS CONTROLLER; é!COCKPIT version *)
RS485BusController.Init(
	StartupDelay := T#5S,				(* Time to wait after startup to start using the bus, prevents boot delay issues when RS485 are not ready yet on startup *)		
	SilenceTime := T#50MS,				(* Silence time between two requests, important to not get faulty data on bus *)
	BusTrigger := ADR(Trigger),			(* Pointer to the bool used to initiate bus requests *)
	BusData := ADR(RtuResponse.awData),	(* Pointer to the array containing the bus response data *)
	BusError := ADR(ModbusMaster.xError)(* Pointer to the bus error bool *)
);

RS485BusController.RegisterDevice(device := FB_RS485_EASTRON_SDM220_1);
RS485BusController.RegisterDevice(device := FB_RS485_ESERA_1WIRE_GATEWAY_MQTT_HOME);
RS485BusController.RegisterDevice(device := FB_RS485_DUCO_DUCOBOX_HOME);

(* INIT RS485 DEVICE STUFF *)
FB_RS485_EASTRON_SDM220_1.InitRS485(
	Data1PollingInterval := T#10S,		(* Polling interval for data array 1 *)				
	Data2PollingInterval := T#20S,		(* Polling interval for data array 2 *)			
	Data3PollingInterval := T#30S,		(* Polling interval for data array 3 *)			
	DeviceAddress := 1					(* Device address of the modbus device *)			
);

FB_RS485_EASTRON_SDM220_1.InitMqtt(
	MQTTPublishPrefix:= ADR(MqttVariables.MqttPubRS485Prefix),						(* pointer to string prefix for the mqtt publish topic *)
	pMqttPublishQueue := ADR(MqttVariables.fbMqttPublishQueue)		(* pointer to MqttPublishQueue to send a new Mqtt event *)
);

FB_RS485_ESERA_1WIRE_GATEWAY_MQTT_HOME.InitRS485(
	DeviceAddress := 2
);

FB_RS485_ESERA_1WIRE_GATEWAY_MQTT_HOME.InitMqtt(
	MQTTPublishPrefix:= ADR(MqttVariables.MqttPubRS485Prefix),	
	pMqttPublishQueue := ADR(MqttVariables.fbMqttPublishQueue)
);

(* ENABLE OWD DEVICES ON ESARE GATEWAY *)
FB_RS485_ESERA_1WIRE_GATEWAY_MQTT_HOME.EnableOwd(
	OwdNumber := 1,
	DataPollingInterval := T#2M
);

FB_RS485_ESERA_1WIRE_GATEWAY_MQTT_HOME.EnableOwd(
	OwdNumber := 2,
	DataPollingInterval := T#2M
);

FB_RS485_DUCO_DUCOBOX_HOME.InitRS485(
	DataPollingInterval := T#3S,		(* Polling interval for data array *)				
	DeviceAddress := 3,					(* Device address of the modbus device *)
);

// Nodes: valves for example
FB_RS485_DUCO_DUCOBOX_HOME.AddNode(
	DataPollingInterval := T#15S
);
FB_RS485_DUCO_DUCOBOX_HOME.AddNode(
	DataPollingInterval := T#15S
);

FB_RS485_DUCO_DUCOBOX_HOME.InitMqtt(
	MQTTPublishPrefix:= ADR(MqttVariables.MqttPubRS485Prefix),
	MQTTSubscribePrefix:= ADR(MqttVariables.MqttSubRS485Prefix),
	pMqttPublishQueue := ADR(MqttVariables.fbMqttPublishQueue),	
	pMqttCallbackCollector := ADR(MqttVariables.collector_FB_RS485_MQTT)
);


END_IF
END_ACTION

ACTION RS485_RUN:
(* CODESYS 3S Version version*)
(*
IF(NOT xComPortOpen AND NOT xComPortError) THEN
    hComPort := SysCom.SysComOpen2( pSettings := ADR(stComPortSettings), pSettingsEx := 0, pResult := ADR(rtsResult));     
    xComPortError := (hComPort = RTS_INVALID_HANDLE OR rtsResult <> 0);
    xComPortOpen := NOT xComPortError;
END_IF


IF xComPortOpen THEN
	fbModbusRequest.modbusCommand.uiFunctionCode := RS485BusController.ActiveRtuQuery.FunctionCode;
    fbModbusRequest.modbusCommand.uiReadOffset := RS485BusController.ActiveRtuQuery.ReadAddress;	
    fbModbusRequest.modbusCommand.uiReadLen :=RS485BusController.ActiveRtuQuery.ReadQuantity;	   
    fbModbusRequest.pRecvData := ADR(awReadBuffer);
    fbModbusRequest.pSendData := ADR(awWriteBuffer);        
    fbModbusRequest.tResponseTimeout := T#1S;
	fbModbusRequest.transmission := MB_Transmission.RTU;
    fbModbusRequest(
        hComPort := hComPort,
        xExecute := Trigger,
        usiSlaveAddr := RS485BusController.ActiveRtuQuery.DeviceId,		
        byModbusError => eComError);
		
END_IF
*)
	
(* é!COCKPIT version*)
RtuQuery.bUnitId := RS485BusController.ActiveRtuQuery.DeviceId;	
RtuQuery.bFunctionCode := RS485BusController.ActiveRtuQuery.FunctionCode;	
RtuQuery.uiReadAddress := RS485BusController.ActiveRtuQuery.ReadAddress;	
RtuQuery.uiReadQuantity := RS485BusController.ActiveRtuQuery.ReadQuantity;
ModbusMaster(
	I_Port := IoConfig_Globals.COM1,
	utQuery:= RtuQuery,
	xTrigger := Trigger,
	utResponse:= RtuResponse);


(* Shared variables for é!COCKPIT and CODESYS 3S Version *)
RS485BusController();

(* RS485 devices *)
FB_RS485_EASTRON_SDM220_1();
FB_RS485_ESERA_1WIRE_GATEWAY_MQTT_HOME();
FB_RS485_DUCO_DUCOBOX_HOME();
END_ACTION

END_PROGRAM

// RS485/FB_RS485_BUSCONTROLLER
FUNCTION_BLOCK FB_RS485_BUSCONTROLLER
VAR_OUTPUT
	///Set this to True by default at startup to allow for some RS485 devices to boot up at power interuptions	
	BusOcupied: BOOL := TRUE;
END_VAR
VAR
	/// Amount of time that should be waited on PLC startup to start using the RS485 bus
	StartupDelay: TIME := TIME#5s0ms;
	/// This is the silence time between two requests
	SilenceTime: TIME := TIME#20ms;
	///Used to detect startup
	Startup: BOOL := TRUE;
	/// To manage silence time and startup delay
	tonDelay: TON;
	///collection of devices on the bus
	devices: ARRAY[0..31] OF RS485Device;
	///total number of devices registred on the bus
	devicesCount: INT := 0;
	///index of the active device on the bus
	selectedDevice: INT := 0;
	deviceActive: BOOL;
	loopCounter: INT;
	ActiveRtuQuery: RS485_RtuQuery;
	BusTrigger: POINTER TO BOOL;
	QueryReady: Standard.F_TRIG;
	BusData: POINTER TO ARRAY[0..124] OF WORD;
	BusError: POINTER TO BOOL;
	exc: __SYSTEM.ExceptionCode;
END_VAR

IF Startup THEN
	tonDelay.PT := StartupDelay;
	tonDelay.IN := TRUE;
	Startup := FALSE;
END_IF

QueryReady(CLK := BusTrigger^);
BusOcupied := NOT(tonDelay.Q);
tonDelay();

// check if there's a device that requires bus time and if so, launch the query
IF busOcupied = FALSE AND deviceActive = FALSE AND devicesCount <> 0 AND NOT QueryReady.Q THEN
	FOR loopCounter := 0 TO devicesCount - 1 DO
		IF deviceActive = FALSE AND devices[loopCounter].RequestBusTime() THEN
			selectedDevice := loopCounter;
			THIS^.SetBusOccupied();
			ActiveRtuQuery := devices[selectedDevice].GetRtuQuery();
			BusTrigger^ := TRUE;
			EXIT;
		END_IF
	END_FOR;
END_IF

//watch the trigger, when completed call the FB with the data, release the bus
IF QueryReady.Q THEN
	devices[selectedDevice].ProcessDataArray(BusError, BusData);
	THIS^.ReleaseBus();
END_IF


//let the busdevices to their work
//FOR loopCounter := 0 TO devicesCount - 1 DO
//	devices[loopCounter]();
// END_FOR;

METHOD Init
VAR_INPUT
	/// Amount of time that should be waited on PLC startup to start using the RS485 bus, can prevent errors due to devices not booted up yet
	StartupDelay: TIME;
	/// This is the silence time between two requests
	SilenceTime: TIME;
	///pointer to the bool that controls triggering busrequests
	BusTrigger: POINTER TO BOOL;
	BusData: POINTER TO ARRAY[0..124] OF WORD;
	BusError: POINTER TO BOOL;
END_VAR
THIS^.StartupDelay := StartupDelay;
THIS^.SilenceTime := SilenceTime;
THIS^.BusTrigger := BusTrigger;
THIS^.BusData := BusData;
THIS^.BusError := BusError;
END_METHOD

METHOD RegisterDevice
VAR_INPUT
	device: RS485Device;
END_VAR
IF devicesCount <> 32 THEN
	devices[devicesCount] := device;
	devicesCount := devicesCount + 1;
END_IF
END_METHOD

METHOD PRIVATE ReleaseBus
// Start a timer to release the bus
THIS^.tonDelay.PT := THIS^.SilenceTime;
THIS^.tonDelay.IN := TRUE;
THIS^.deviceActive := FALSE;
END_METHOD

METHOD PRIVATE SetBusOccupied
THIS^.tonDelay.IN := FALSE;
THIS^.deviceActive := TRUE;
END_METHOD

END_FUNCTION_BLOCK

// RS485/RS485Device
INTERFACE RS485Device

METHOD GetRtuQuery : RS485_RtuQuery
END_METHOD

METHOD ProcessDataArray
VAR_INPUT
	Error: POINTER TO BOOL;
	Data: POINTER TO ARRAY[0..124] OF WORD;
END_VAR
END_METHOD

METHOD RequestBusTime : BOOL
END_METHOD

END_INTERFACE

// FB_RS485_EASTRON_SDM220_MQTT
{attribute 'reflection' := ''}
FUNCTION_BLOCK FB_RS485_EASTRON_SDM220_MQTT IMPLEMENTS RS485Device
VAR_OUTPUT
	VOLTAGE: REAL := 0;
	CURRENT: REAL := 0;
	ACTIVEPOWER: REAL := 0;
	APPARENT_POWER: REAL := 0;
	REACTIVE_POWER: REAL := 0;
	POWER_FACTOR: REAL := 0;
	PHASE_ANGLE: REAL := 0;
	DataAvailable1: BOOL := FALSE;
	Error1: BOOL := FALSE;
	FREQUENCY: REAL := 0;
	IMPORT_ACTIVE_ENERGY: REAL := 0;
	EXPORT_ACTIVE_ENERGY: REAL := 0;
	IMPORT_REACTIVE_ENERGY: REAL := 0;
	EXPORT_REACTIVE_ENERGY: REAL := 0;
	DataAvailable2: BOOL := FALSE;
	Error2: BOOL := FALSE;
	TOTAL_ACTIVE_ENERGY: REAL := 0;
	TOTAL_REACTIVE_ENERGY: REAL := 0;
	DataAvailable3: BOOL := FALSE;
	Error3: BOOL := FALSE;
END_VAR
VAR
	/// object's full instance name 
	{attribute 'noinit'}
	{attribute 'instance-path' := ''}
	InstanceName: STRING;
	Startup: BOOL := TRUE;
	InitMqttDone: BOOL;
	MqttPublishTopicPrefix: POINTER TO STRING;
	MqttPublishTopicSuffix: STRING(50);
	pMqttPublishQueue: POINTER TO FB_MqttPublishQueue;
	InitRS485Done: BOOL := FALSE;
	ActiveDevice: BOOL := FALSE;
	ActiveRtuQuery: INT := 0;
	Data1RtuQuery: RS485_RtuQuery := (FunctionCode := 4, ReadAddress := 0, ReadQuantity := 40);
	Update1: BOOL := FALSE;
	timerData1: TON;
	Data2RtuQuery: RS485_RtuQuery := (FunctionCode := 4, ReadAddress := 70, ReadQuantity := 10);
	Update2: BOOL := FALSE;
	timerData2: TON;
	Data3RtuQuery: RS485_RtuQuery := (FunctionCode := 4, ReadAddress := 342, ReadQuantity := 4);
	Update3: BOOL := FALSE;
	timerData3: TON;
END_VAR

timerData1();
timerData2();
timerData3();

IF Update1 THEN
	Update1 := FALSE;
	DataAvailable1 := TRUE;
	
	IF InitMqttDone THEN
		pMqttPublishQueue^.AddMessage(
			Payload := REAL_TO_STRING(VOLTAGE),
			Topic := CONCAT(CONCAT(MqttPublishTopicPrefix^, MqttPublishTopicSuffix), '/VOLT' ),
			Qos := MQTT.QoS.ExactlyOnce,
			MqttRetain := FALSE
		);
		pMqttPublishQueue^.AddMessage(
			Payload := REAL_TO_STRING(CURRENT),
			Topic := CONCAT(CONCAT(MqttPublishTopicPrefix^, MqttPublishTopicSuffix), '/CURR' ),
			Qos := MQTT.QoS.ExactlyOnce,
			MqttRetain := FALSE
		);	
		pMqttPublishQueue^.AddMessage(
			Payload := REAL_TO_STRING(ACTIVEPOWER),
			Topic := CONCAT(CONCAT(MqttPublishTopicPrefix^, MqttPublishTopicSuffix), '/ACTP' ),
			Qos := MQTT.QoS.ExactlyOnce,
			MqttRetain := FALSE
		);
		pMqttPublishQueue^.AddMessage(
			Payload := REAL_TO_STRING(APPARENT_POWER),
			Topic := CONCAT(CONCAT(MqttPublishTopicPrefix^, MqttPublishTopicSuffix), '/APPP' ),
			Qos := MQTT.QoS.ExactlyOnce,
			MqttRetain := FALSE
		);
		pMqttPublishQueue^.AddMessage(
			Payload := REAL_TO_STRING(REACTIVE_POWER),
			Topic := CONCAT(CONCAT(MqttPublishTopicPrefix^, MqttPublishTopicSuffix), '/REAP' ),
			Qos := MQTT.QoS.ExactlyOnce,
			MqttRetain := FALSE
		);
		pMqttPublishQueue^.AddMessage(
			Payload := REAL_TO_STRING(POWER_FACTOR),
			Topic := CONCAT(CONCAT(MqttPublishTopicPrefix^, MqttPublishTopicSuffix), '/POWF' ),
			Qos := MQTT.QoS.ExactlyOnce,
			MqttRetain := FALSE
		);
		pMqttPublishQueue^.AddMessage(
			Payload := REAL_TO_STRING(PHASE_ANGLE),
			Topic := CONCAT(CONCAT(MqttPublishTopicPrefix^, MqttPublishTopicSuffix), '/PHAA' ),
			Qos := MQTT.QoS.ExactlyOnce,
			MqttRetain := FALSE
		);
	END_IF
END_IF

IF Update2 THEN
	Update2 := FALSE;
	DataAvailable2 := TRUE;
	
	IF InitMqttDone THEN
		pMqttPublishQueue^.AddMessage(
			Payload := REAL_TO_STRING(FREQUENCY),
			Topic := CONCAT(CONCAT(MqttPublishTopicPrefix^, MqttPublishTopicSuffix), '/FREQ' ),
			Qos := MQTT.QoS.ExactlyOnce,
			MqttRetain := FALSE
		);
		pMqttPublishQueue^.AddMessage(
			Payload := REAL_TO_STRING(IMPORT_ACTIVE_ENERGY),
			Topic := CONCAT(CONCAT(MqttPublishTopicPrefix^, MqttPublishTopicSuffix), '/IMAE' ),
			Qos := MQTT.QoS.ExactlyOnce,
			MqttRetain := FALSE
		);
		pMqttPublishQueue^.AddMessage(
			Payload := REAL_TO_STRING(EXPORT_ACTIVE_ENERGY),
			Topic := CONCAT(CONCAT(MqttPublishTopicPrefix^, MqttPublishTopicSuffix), '/EXAE' ),
			Qos := MQTT.QoS.ExactlyOnce,
			MqttRetain := FALSE
		);
		pMqttPublishQueue^.AddMessage(
			Payload := REAL_TO_STRING(IMPORT_REACTIVE_ENERGY),
			Topic := CONCAT(CONCAT(MqttPublishTopicPrefix^, MqttPublishTopicSuffix), '/IMRE' ),
			Qos := MQTT.QoS.ExactlyOnce,
			MqttRetain := FALSE
		);
		pMqttPublishQueue^.AddMessage(
			Payload := REAL_TO_STRING(EXPORT_REACTIVE_ENERGY),
			Topic := CONCAT(CONCAT(MqttPublishTopicPrefix^, MqttPublishTopicSuffix), '/EXRE' ),
			Qos := MQTT.QoS.ExactlyOnce,
			MqttRetain := FALSE
		);
	END_IF
END_IF

IF Update3 THEN
	Update3 := FALSE;	
	DataAvailable3 := TRUE;
	
	IF InitMqttDone THEN
		pMqttPublishQueue^.AddMessage(
			Payload := REAL_TO_STRING(TOTAL_ACTIVE_ENERGY),
			Topic := CONCAT(CONCAT(MqttPublishTopicPrefix^, MqttPublishTopicSuffix), '/TOTAE' ),
			Qos := MQTT.QoS.ExactlyOnce,
			MqttRetain := FALSE
		);
		pMqttPublishQueue^.AddMessage(
			Payload := REAL_TO_STRING(TOTAL_REACTIVE_ENERGY),
			Topic := CONCAT(CONCAT(MqttPublishTopicPrefix^, MqttPublishTopicSuffix), '/TOTRE' ),
			Qos := MQTT.QoS.ExactlyOnce,
			MqttRetain := FALSE
		);
	END_IF
END_IF

METHOD GetRtuQuery : RS485_RtuQuery
IF timerData1.Q THEN
	THIS^.timerData1.IN := FALSE;
	THIS^.ActiveRtuQuery := 1;
	GetRtuQuery := THIS^.Data1RtuQuery;
ELSIF timerData2.Q THEN
	THIS^.timerData2.IN := FALSE;
	THIS^.ActiveRtuQuery := 2;
	GetRtuQuery := THIS^.Data2RtuQuery;
ELSIF timerData3.Q THEN
	THIS^.timerData3.IN := FALSE;
	THIS^.ActiveRtuQuery := 3;
	GetRtuQuery := THIS^.Data3RtuQuery;	
END_IF
END_METHOD

METHOD InitMqtt
VAR_INPUT
	MQTTPublishPrefix: POINTER TO STRING;
	pMqttPublishQueue: POINTER TO FB_MqttPublishQueue;
END_VAR
VAR
	InstanceNamePt: POINTER TO STRING;
END_VAR
THIS^.pMqttPublishQueue := pMqttPublishQueue;
THIS^.MqttPublishTopicPrefix := MQTTPublishPrefix;

InstanceNamePt := CommonTypesAndFunctions.FindLastDot(ADR(THIS^.InstanceName)) + 1;
THIS^.MqttPublishTopicSuffix := InstanceNamePt^;

THIS^.InitMqttDone := TRUE;
END_METHOD

METHOD InitRS485
VAR_INPUT
	Data1PollingInterval: TIME;
	Data2PollingInterval: TIME;
	Data3PollingInterval: TIME;
	DeviceAddress: BYTE;
END_VAR
THIS^.timerData1.PT := Data1PollingInterval;
THIS^.timerData2.PT := Data2PollingInterval;
THIS^.timerData3.PT := Data3PollingInterval;

THIS^.Data1RtuQuery.DeviceId := DeviceAddress;
THIS^.Data2RtuQuery.DeviceId := DeviceAddress;
THIS^.Data3RtuQuery.DeviceId := DeviceAddress;

THIS^.timerData1.IN := TRUE;
THIS^.timerData2.IN := TRUE;
THIS^.timerData3.IN := TRUE;

THIS^.InitRS485Done := TRUE;
END_METHOD

METHOD ProcessDataArray
VAR_INPUT
	Error: POINTER TO BOOL;
	Data: POINTER TO ARRAY[0..124] OF WORD;
END_VAR
IF Error^ THEN
	PubMqttMessage(Suffix := '/availability', Data := 'offline');
ELSE
	PubMqttMessage(Suffix := '/availability', Data := 'online');
END_IF

IF ActiveRtuQuery = 1 THEN
	THIS^.Error1 := Error^;
	THIS^.timerData1.IN := TRUE;
	IF NOT Error^ THEN
		THIS^.VOLTAGE := SwapWordsToReal(Data^[0], Data^[1]);
		THIS^.CURRENT := SwapWordsToReal(Data^[6], Data^[7]);
		THIS^.ACTIVEPOWER := SwapWordsToReal(Data^[12], Data^[13]);
		THIS^.APPARENT_POWER := SwapWordsToReal(Data^[18], Data^[19]);
		THIS^.REACTIVE_POWER := SwapWordsToReal(Data^[24], Data^[25]);
		THIS^.POWER_FACTOR := SwapWordsToReal(Data^[30], Data^[31]);
		THIS^.PHASE_ANGLE := SwapWordsToReal(Data^[36], Data^[37]);
		THIS^.Update1 := TRUE;
	END_IF
ELSIF ActiveRtuQuery = 2 THEN
	THIS^.Error2:= Error^;
	THIS^.timerData2.IN := TRUE;
	IF NOT Error^ THEN		
		THIS^.FREQUENCY := SwapWordsToReal(Data^[0], Data^[1]);
		THIS^.IMPORT_ACTIVE_ENERGY := SwapWordsToReal(Data^[2], Data^[3]);
		THIS^.EXPORT_ACTIVE_ENERGY := SwapWordsToReal(Data^[4], Data^[5]);
		THIS^.IMPORT_REACTIVE_ENERGY := SwapWordsToReal(Data^[6], Data^[7]);
		THIS^.EXPORT_REACTIVE_ENERGY := SwapWordsToReal(Data^[8], Data^[9]);
		THIS^.Update2 := TRUE;
	END_IF
ELSIF ActiveRtuQuery = 3 THEN
	THIS^.Error3 := Error^;
	THIS^.timerData3.IN := TRUE;
	IF NOT Error^ THEN
		THIS^.TOTAL_ACTIVE_ENERGY := SwapWordsToReal(Data^[0], Data^[1]);
		THIS^.TOTAL_REACTIVE_ENERGY := SwapWordsToReal(Data^[2], Data^[3]);
		THIS^.Update3 := TRUE;
	END_IF	
END_IF

ActiveRtuQuery := 0;
ActiveDevice := FALSE;
END_METHOD

METHOD PubMqttMessage
VAR_INPUT
	Suffix: STRING(100);
	Data: STRING(100);
END_VAR
IF InitMqttDone THEN
		pMqttPublishQueue^.AddMessage(
			Payload := Data,
			Topic := CONCAT(CONCAT(MqttPublishTopicPrefix^, MqttPublishTopicSuffix), Suffix ),
			Qos := MQTT.QoS.ExactlyOnce,
			MqttRetain := FALSE
		);
END_IF
END_METHOD

METHOD RequestBusTime : BOOL
IF NOT InitRS485Done THEN	
	RequestBusTime := FALSE;	
ELSIF timerData1.Q OR timerData2.Q OR timerData3.Q THEN
	RequestBusTime := TRUE;	
ELSE
	RequestBusTime := FALSE;		
END_IF
END_METHOD

END_FUNCTION_BLOCK

// SwapWordsToReal
FUNCTION SwapWordsToReal : REAL
VAR_INPUT
	wHi: WORD;
	wLo: WORD;
END_VAR
VAR
	dwVar: DWORD;
	pt_REAL: POINTER TO REAL;
END_VAR

dwVar := SHL(WORD_TO_DWORD(wHi),16) OR WORD_TO_DWORD(wLo);
pt_REAL := ADR(dwVar);
SwapWordsToReal := pt_REAL^;

END_FUNCTION

// FB_RS485_ESERA_1WIRE_GATEWAY_MQTT
{attribute 'reflection' := ''}
FUNCTION_BLOCK FB_RS485_ESERA_1WIRE_GATEWAY_MQTT IMPLEMENTS RS485Device
VAR
	/// object's full instance name 
	{attribute 'noinit'}
	{attribute 'instance-path' := ''}
	InstanceName: STRING;
	InitRS485Done: BOOL := FALSE;
	DeviceAddress: BYTE;
	OwdDevices: ARRAY[1..30] OF FB_RS485_ESERA_OWD_MQTT;
	ActiveDevice: BOOL := FALSE;
	ActiveOwd: UINT := 0;
	loopCounter: UINT;
	timerData: TON;
END_VAR

timerData();

FOR loopCounter := 1 TO 30 DO
	OwdDevices[loopCounter]();
END_FOR

METHOD EnableOwd : BOOL
VAR_INPUT
	OwdNumber: UINT;
	DataPollingInterval: TIME;
END_VAR
THIS^.OwdDevices[OwdNumber].InitOwd(
	DeviceAddress := THIS^.DeviceAddress,
	OwdNumber := OwdNumber,
	DataPollingInterval := DataPollingInterval
);
END_METHOD

METHOD GetRtuQuery : RS485_RtuQuery
IF timerData.Q THEN
	THIS^.timerData.IN := FALSE;
	GetRtuQuery := THIS^.OwdDevices[ActiveOwd].GetRtuQuery();	
END_IF
END_METHOD

METHOD InitMqtt
VAR_INPUT
	MQTTPublishPrefix: POINTER TO STRING;
	pMqttPublishQueue: POINTER TO FB_MqttPublishQueue;
END_VAR
VAR
	InstanceNamePt: POINTER TO STRING;
END_VAR
InstanceNamePt := CommonTypesAndFunctions.FindLastDot(ADR(THIS^.InstanceName)) + 1;

FOR loopCounter := 1 TO 30 DO
		OwdDevices[loopCounter].InitMqtt(
			MQTTPublishPrefix := MQTTPublishPrefix,
			MqttPublishTopicSuffix := InstanceNamePt^,
			pMqttPublishQueue := pMqttPublishQueue
		);
END_FOR
END_METHOD

METHOD InitRS485
VAR_INPUT
	DeviceAddress: BYTE;
END_VAR
THIS^.DeviceAddress := DeviceAddress;
THIS^.timerData.PT := T#250MS;
THIS^.timerData.IN := TRUE;
THIS^.InitRS485Done := TRUE;
END_METHOD

METHOD ProcessDataArray
VAR_INPUT
	Error: POINTER TO BOOL;
	Data: POINTER TO ARRAY[0..124] OF WORD;
END_VAR
THIS^.OwdDevices[ActiveOwd].ProcessDataArray(
	Data := Data,
	Error := Error
);
THIS^.ActiveOwd := 0;
THIS^.timerData.IN := TRUE;
END_METHOD

METHOD RequestBusTime : BOOL
IF NOT InitRS485Done OR NOT timerData.Q THEN	
	RequestBusTime := FALSE;
ELSE
	FOR loopCounter := 1 TO 30 DO
		IF OwdDevices[loopCounter].RequestBusTime() AND RequestBusTime = FALSE THEN
			THIS^.ActiveOwd := loopCounter;
			RequestBusTime := TRUE;			
		END_IF
	END_FOR
END_IF
END_METHOD

END_FUNCTION_BLOCK

// FB_RS485_ESERA_OWD_MQTT
FUNCTION_BLOCK FB_RS485_ESERA_OWD_MQTT
VAR_OUTPUT
	OWD_VOLTAGE: REAL := 0;
	TEMPERATURE: REAL := 0;
	HUMIDITY: REAL := 0;
	DEW_POINT: REAL := 0;
	AIR_QUALITY: REAL := 0;
	BRIGHTNESS: REAL := 0;
	DataAvailable: BOOL := FALSE;
	Error: BOOL := FALSE;
END_VAR
VAR
	OwdNumber: UINT;
	InitMqttDone: BOOL;
	MqttPublishTopicPrefix: POINTER TO STRING;
	MqttPublishTopicSuffix: STRING(50);
	pMqttPublishQueue: POINTER TO FB_MqttPublishQueue;
	InitOwdDone: BOOL := FALSE;
	timerData: TON;
	RtuQuery: RS485_RtuQuery := (FunctionCode := 3, ReadAddress := 100, ReadQuantity := 17);
END_VAR

timerData();

METHOD GetRtuQuery : RS485_RtuQuery
IF timerData.Q THEN
	THIS^.timerData.IN := FALSE;
	GetRtuQuery := THIS^.RtuQuery;	
END_IF
END_METHOD

METHOD InitMqtt
VAR_INPUT
	MQTTPublishPrefix: POINTER TO STRING;
	MqttPublishTopicSuffix: STRING(255);
	pMqttPublishQueue: POINTER TO FB_MqttPublishQueue;
END_VAR
THIS^.MqttPublishTopicPrefix := MQTTPublishPrefix;
THIS^.MqttPublishTopicSuffix := MqttPublishTopicSuffix;
THIS^.pMqttPublishQueue := pMqttPublishQueue;

THIS^.InitMqttDone := TRUE;
END_METHOD

METHOD InitOwd
VAR_INPUT
	DeviceAddress: BYTE;
	OwdNumber: UINT;
	DataPollingInterval: TIME;
END_VAR
THIS^.RtuQuery.DeviceId := DeviceAddress;
THIS^.RtuQuery.ReadAddress := OwdNumber * 100;
THIS^.timerData.PT := DataPollingInterval;
THIS^.OwdNumber := OwdNumber;

THIS^.timerData.IN := TRUE;

THIS^.InitOwdDone := TRUE;
END_METHOD

METHOD ProcessAirQuality
VAR_INPUT
	Data: WORD;
END_VAR
THIS^.AIR_QUALITY := WORD_TO_REAL(Data) / 100;
PubMqttMessage(Suffix := '/AIRQ', Data := REAL_TO_STRING(AIR_QUALITY));
END_METHOD

METHOD ProcessBrigthness
VAR_INPUT
	Data: WORD;
END_VAR
THIS^.BRIGHTNESS := WORD_TO_REAL(Data) / 100;
PubMqttMessage(Suffix := '/BNESS', Data := REAL_TO_STRING(BRIGHTNESS));
END_METHOD

METHOD ProcessDataArray
VAR_INPUT
	Error: POINTER TO BOOL;
	Data: POINTER TO ARRAY[0..124] OF WORD;
END_VAR
THIS^.timerData.IN := TRUE;

IF WORD_TO_INT(Data^[12]) <> 0 OR Error^ THEN
	THIS^.Error := TRUE;
	PubMqttMessage(Suffix := '/availability', Data := 'offline');
ELSE 	
	THIS^.Error := FALSE;
	THIS^.DataAvailable := TRUE;
	PubMqttMessage(Suffix := '/availability', Data := 'online');
END_IF

// Data handling
IF NOT Error^ AND WORD_TO_INT(Data^[12]) = 0 THEN
	IF Data^[16] = 11151 OR Data^[16] = 11152 THEN // Temperature, humidity & air quality
		ProcessTemperature(Data^[0]);		
		ProcessOwdVoltage(Data^[2]);
		ProcessHumidity(Data^[4]);
		ProcessDewPoint(Data^[6]);
		ProcessAirQuality(Data^[8]);
	ELSIF Data^[16] = 11102 OR Data^[16] = 11113 OR Data^[16] = 11120 OR Data^[16] = 11148 OR Data^[16] = 11150 OR Data^[16] = 11160 THEN // Temperature, humidity
		ProcessTemperature(Data^[0]);		
		ProcessOwdVoltage(Data^[2]);
		ProcessHumidity(Data^[4]);
		ProcessDewPoint(Data^[6]);
	ELSIF Data^[16] = 11121 OR Data^[16] = 11132 OR Data^[16] = 11134 OR Data^[16] = 11135 THEN // Temperature, humidity, brightness
		ProcessTemperature(Data^[0]);		
		ProcessOwdVoltage(Data^[2]);
		ProcessHumidity(Data^[4]);
		ProcessDewPoint(Data^[6]);
		ProcessBrigthness(Data^[8]);
	ELSIF Data^[16] = 1820  THEN // Temperature DS18B20
        ProcessTemperature(Data^[0]);
	END_IF		
END_IF
END_METHOD

METHOD ProcessDewPoint
VAR_INPUT
	Data: WORD;
END_VAR
THIS^.DEW_POINT := WORD_TO_REAL(Data) / 100;
PubMqttMessage(Suffix := '/DEWP', Data := REAL_TO_STRING(DEW_POINT));
END_METHOD

METHOD ProcessHumidity
VAR_INPUT
	Data: WORD;
END_VAR
THIS^.HUMIDITY := WORD_TO_REAL(Data) / 100;
PubMqttMessage(Suffix := '/HUM', Data := REAL_TO_STRING(HUMIDITY));
END_METHOD

METHOD ProcessOwdVoltage
VAR_INPUT
	Data: WORD;
END_VAR
THIS^.OWD_VOLTAGE := WORD_TO_REAL(Data) / 100;
PubMqttMessage(Suffix := '/OWDV', Data := REAL_TO_STRING(OWD_VOLTAGE));
END_METHOD

METHOD ProcessTemperature
VAR_INPUT
	Data: WORD;
END_VAR
THIS^.TEMPERATURE := WORD_TO_REAL(Data) / 100;
PubMqttMessage(Suffix := '/TEMP', Data := REAL_TO_STRING(TEMPERATURE));
END_METHOD

METHOD PubMqttMessage
VAR_INPUT
	Suffix: STRING(100);
	Data: STRING(100);
END_VAR
IF InitMqttDone THEN
		pMqttPublishQueue^.AddMessage(
			Payload := Data,
			Topic := CONCAT(CONCAT(CONCAT(CONCAT(MqttPublishTopicPrefix^, MqttPublishTopicSuffix), '/OWD/'), UINT_TO_STRING(OwdNumber)), Suffix ),
			Qos := MQTT.QoS.ExactlyOnce,
			MqttRetain := FALSE
		);
END_IF
END_METHOD

METHOD RequestBusTime : BOOL
IF NOT InitOwdDone THEN	
	RequestBusTime := FALSE;	
ELSIF timerData.Q THEN
	RequestBusTime := TRUE;
ELSE
	RequestBusTime := FALSE;	
END_IF
END_METHOD

END_FUNCTION_BLOCK

// FB_RS485_DUCO_DUCOBOX_MQTT
{attribute 'reflection' := ''}
FUNCTION_BLOCK FB_RS485_DUCO_DUCOBOX_MQTT IMPLEMENTS RS485Device, MQTT.MQTT_SUBSCRIBE_CALLBACK
VAR_OUTPUT
	ACTIVEPOWER: REAL := 0;
	DataAvailable: BOOL := FALSE;
	Error: BOOL := FALSE;
END_VAR
VAR
	/// object's full instance name 
	{attribute 'instance-path' := ''}
	{attribute 'noinit' := ''}
	InstanceName: STRING;
	Startup: BOOL := TRUE;
	InitMqttDone: BOOL;
	MqttPublishTopicPrefix: POINTER TO STRING;
	MqttPublishTopicSuffix: STRING(50);
	MQTTSubscribeTopic: STRING(50);
	pMqttPublishQueue: POINTER TO FB_MqttPublishQueue;
	InitRS485Done: BOOL := FALSE;
	timerData: TON;
	isDataUpdated: BOOL := FALSE;
	Nodes: ARRAY[2..30] OF FB_RS485_DUCO_DUCOBOX_NODE_MQTT;
	NodePointer: UINT := 2;
	ActiveNode: INT := 0;
	loopCounter: INT;
	ReadMasterUnitQuery: RS485_RtuQuery := (FunctionCode := 4, ReadAddress := 10, ReadQuantity := 6);
	WriteQueryReady: BOOL := FALSE;
	WriteQueryBeingExecuted: BOOL := FALSE;
	WriteQuerySuffix: STRING;
	WriteQueryPayload: STRING;
	WriteQuery: RS485_RtuQuery := (FunctionCode := 6, WriteQuantity := 1);
END_VAR

timerData();

FOR loopCounter := 2 TO 30 DO
	Nodes[loopCounter]();
END_FOR

METHOD AddNode : BOOL
VAR_INPUT
	DataPollingInterval: TIME;
END_VAR
THIS^.Nodes[NodePointer].InitNode(
	DeviceAddress := THIS^.ReadMasterUnitQuery.DeviceId,
	NodeNumber := NodePointer -1,
	DataPollingInterval := DataPollingInterval
);

NodePointer := NodePointer + 1;
END_METHOD

METHOD GetRtuQuery : RS485_RtuQuery
IF WriteQueryReady THEN
	GetRtuQuery := THIS^.WriteQuery;
	WriteQueryBeingExecuted := TRUE;
// master
ELSIF ActiveNode = 1 THEN
	THIS^.timerData.IN := FALSE;
	GetRtuQuery := THIS^.ReadMasterUnitQuery;
// other nodes
ELSIF ActiveNode > 1 THEN
	GetRtuQuery := THIS^.Nodes[ActiveNode].GetRtuQuery();	
END_IF
END_METHOD

METHOD InitMqtt
VAR_INPUT
	MQTTPublishPrefix: POINTER TO STRING;
	MQTTSubscribePrefix: POINTER TO STRING;
	pMqttPublishQueue: POINTER TO FB_MqttPublishQueue;
	pMqttCallbackCollector: POINTER TO MQTT.CallbackCollector;
END_VAR
VAR
	InstanceNamePt: POINTER TO STRING;
END_VAR
THIS^.pMqttPublishQueue := pMqttPublishQueue;
THIS^.MqttPublishTopicPrefix := MQTTPublishPrefix;

InstanceNamePt := CommonTypesAndFunctions.FindLastDot(ADR(THIS^.InstanceName)) + 1;
THIS^.MqttPublishTopicSuffix := InstanceNamePt^;
THIS^.MQTTSubscribeTopic := CONCAT(MQTTSubscribePrefix^ ,THIS^.MqttPublishTopicSuffix);

// register the FB agains the collector so mqtt events can be received
pMqttCallbackCollector^.put(instance:= THIS^);


FOR loopCounter := 2 TO 30 DO
		Nodes[loopCounter].InitMqtt(
			MQTTPublishPrefix := MQTTPublishPrefix,
			MqttPublishTopicSuffix := InstanceNamePt^,
			pMqttPublishQueue := pMqttPublishQueue
		);
END_FOR

InitMqttDone := TRUE;
END_METHOD

METHOD InitRS485
VAR_INPUT
	DataPollingInterval: TIME;
	DeviceAddress: BYTE;
END_VAR
THIS^.timerData.PT := DataPollingInterval;
THIS^.ReadMasterUnitQuery.DeviceId := DeviceAddress;
THIS^.WriteQuery.DeviceId := DeviceAddress;
THIS^.timerData.IN := TRUE;

THIS^.InitRS485Done := TRUE;
END_METHOD

METHOD ProcessDataArray
VAR_INPUT
	Error: POINTER TO BOOL;
	Data: POINTER TO ARRAY[0..124] OF WORD;
END_VAR
THIS^.Error := Error^;

IF Error^ AND NOT WriteQueryBeingExecuted THEN
	PubMqttMessage(Suffix := '/availability', Data := 'offline');
ELSE
	PubMqttMessage(Suffix := '/availability', Data := 'online');
END_IF

IF WriteQueryBeingExecuted THEN
	WriteQueryReady := FALSE;
	WriteQueryBeingExecuted := FALSE;
	IF NOT Error^ THEN
		PubMqttMessage(Suffix := CONCAT('/', WriteQuerySuffix), Data := WriteQueryPayload);
	END_IF
// data for master unit (= main node)
ELSIF THIS^.ActiveNode = 1 THEN
	THIS^.timerData.IN := TRUE;
	THIS^.ActiveNode := 0;
	
	IF NOT Error^ THEN
 		PubMqttMessage(Suffix := '/1/read/0', Data := WORD_TO_STRING(Data^[0]));
 		PubMqttMessage(Suffix := '/1/read/1', Data := WORD_TO_STRING(Data^[1]));
 		PubMqttMessage(Suffix := '/1/read/2', Data := WORD_TO_STRING(Data^[2]));
 		PubMqttMessage(Suffix := '/1/read/3', Data := WORD_TO_STRING(Data^[3]));
 		PubMqttMessage(Suffix := '/1/read/4', Data := WORD_TO_STRING(Data^[4]));
 		PubMqttMessage(Suffix := '/1/read/5', Data := WORD_TO_STRING(Data^[5]));
	END_IF
// data for nodes
ELSIF THIS^.ActiveNode > 1 THEN	
	THIS^.Nodes[ActiveNode].ProcessDataArray(
		Data := Data,
		Error := Error
	);
	THIS^.ActiveNode := 0;
END_IF
END_METHOD

METHOD PublishReceived : BOOL
VAR_INPUT
	///Collection of recived Data
	Data: MQTT.CALLBACK_DATA;
END_VAR
VAR
	SubTopic: STRING;
	NodeNumber: STRING;
	NodeRegister: STRING;
END_VAR
//first check if Mqtt is initialized, otherwise do nothing
IF NOT(InitMqttDone) THEN
	//mark the interface call from the collector as done
	PublishReceived := TRUE;
//check if the packet is for this FB
ELSIF MQTTSubscribeTopic = LEFT(Data.TopicOut^, LEN(MQTTSubscribeTopic)) THEN
	//mark the interface call from the collector as done
	PublishReceived := TRUE;
	// process the data
	SubTopic := RIGHT(Data.TopicOut^, 9); // 2/write/9 -> 10 chars
	NodeNumber := LEFT(SubTopic, 1);
	NodeRegister := RIGHT(SubTopic, 1);
	
	IF FIND(SubTopic, 'write') > 0 AND
		OSCAT_BASIC.IS_NUM(NodeNumber) AND
		OSCAT_BASIC.IS_NUM(NodeRegister) AND
		OSCAT_BASIC.IS_NUM(Data.PayloadString^) THEN
			WriteQuery.WriteAddress := (STRING_TO_UINT(NodeNumber) * 10) + STRING_TO_UINT(NodeRegister);
			WriteQuery.WriteData[0] := STRING_TO_WORD(Data.PayloadString^);
			WriteQuerySuffix := SubTopic;
			WriteQueryPayload := Data.PayloadString^;
			WriteQueryReady := TRUE;
	END_IF
END_IF
END_METHOD

METHOD PubMqttMessage
VAR_INPUT
	Suffix: STRING(100);
	Data: STRING(100);
END_VAR
IF InitMqttDone THEN
		pMqttPublishQueue^.AddMessage(
			Payload := Data,
			Topic := CONCAT(CONCAT(MqttPublishTopicPrefix^, MqttPublishTopicSuffix), Suffix ),
			Qos := MQTT.QoS.ExactlyOnce,
			MqttRetain := FALSE
		);
END_IF
END_METHOD

METHOD RequestBusTime : BOOL
IF NOT InitRS485Done THEN	
	RequestBusTime := FALSE;
ELSIF WriteQueryReady THEN
	RequestBusTime := TRUE;	
ELSIF timerData.Q THEN // Master node
	RequestBusTime := TRUE;
	THIS^.ActiveNode := 1;
ELSIF NodePointer > 2 THEN// other nodes, if configured
	FOR loopCounter := 2 TO 30 DO
		IF Nodes[loopCounter].RequestBusTime() AND RequestBusTime = FALSE THEN
			THIS^.ActiveNode := loopCounter;
			RequestBusTime := TRUE;	
		END_IF
	END_FOR
ELSE
	RequestBusTime := FALSE;
END_IF
END_METHOD

END_FUNCTION_BLOCK

// FB_RS485_DUCO_DUCOBOX_NODE_MQTT
FUNCTION_BLOCK FB_RS485_DUCO_DUCOBOX_NODE_MQTT
VAR
	NodeNumber: UINT;
	InitMqttDone: BOOL;
	MqttPublishTopicPrefix: POINTER TO STRING;
	MqttPublishTopicSuffix: STRING(51);
	pMqttPublishQueue: POINTER TO FB_MqttPublishQueue;
	NodeInitialized: BOOL := FALSE;
	timerData: TON;
	RtuQueryRead: RS485_RtuQuery := (FunctionCode := 4, ReadAddress := 20, ReadQuantity := 6);
END_VAR

timerData();

METHOD GetRtuQuery : RS485_RtuQuery
IF timerData.Q THEN
	THIS^.timerData.IN := FALSE;
	GetRtuQuery := THIS^.RtuQueryRead;	
END_IF
END_METHOD

METHOD InitMqtt
VAR_INPUT
	MQTTPublishPrefix: POINTER TO STRING;
	MqttPublishTopicSuffix: STRING(255);
	pMqttPublishQueue: POINTER TO FB_MqttPublishQueue;
END_VAR
THIS^.MqttPublishTopicPrefix := MQTTPublishPrefix;
THIS^.MqttPublishTopicSuffix := MqttPublishTopicSuffix;
THIS^.pMqttPublishQueue := pMqttPublishQueue;

THIS^.InitMqttDone := TRUE;
END_METHOD

METHOD InitNode
VAR_INPUT
	DeviceAddress: BYTE;
	NodeNumber: UINT;
	DataPollingInterval: TIME;
END_VAR
THIS^.RtuQueryRead.DeviceId := DeviceAddress;
THIS^.RtuQueryRead.ReadAddress := (NodeNumber * 10) + 10;

THIS^.timerData.PT := DataPollingInterval;
THIS^.NodeNumber := NodeNumber + 1;

THIS^.timerData.IN := TRUE;

THIS^.NodeInitialized := TRUE;
END_METHOD

METHOD ProcessDataArray
VAR_INPUT
	Error: POINTER TO BOOL;
	Data: POINTER TO ARRAY[0..124] OF WORD;
END_VAR
THIS^.timerData.IN := TRUE;

IF NOT Error^ THEN
	PubMqttMessage(Suffix := '/read/0', Data := WORD_TO_STRING(Data^[0]));
	PubMqttMessage(Suffix := '/read/1', Data := WORD_TO_STRING(Data^[1]));
	PubMqttMessage(Suffix := '/read/2', Data := WORD_TO_STRING(Data^[2]));
	PubMqttMessage(Suffix := '/read/3', Data := WORD_TO_STRING(Data^[3]));
	PubMqttMessage(Suffix := '/read/4', Data := WORD_TO_STRING(Data^[4]));
	PubMqttMessage(Suffix := '/read/5', Data := WORD_TO_STRING(Data^[5]));
END_IF
END_METHOD

METHOD PubMqttMessage
VAR_INPUT
	Suffix: STRING(100);
	Data: STRING(100);
END_VAR
IF InitMqttDone THEN
		pMqttPublishQueue^.AddMessage(
			Payload := Data,
			Topic := CONCAT(CONCAT(CONCAT(CONCAT(MqttPublishTopicPrefix^, MqttPublishTopicSuffix), '/'), UINT_TO_STRING(NodeNumber)), Suffix ),
			Qos := MQTT.QoS.ExactlyOnce,
			MqttRetain := FALSE
		);
END_IF
END_METHOD

METHOD RequestBusTime : BOOL
IF NOT NodeInitialized THEN	
	RequestBusTime := FALSE;
ELSIF timerData.Q THEN
	RequestBusTime := TRUE;
ELSE
	RequestBusTime := FALSE;	
END_IF
END_METHOD

END_FUNCTION_BLOCK

// FB_INPUT_BINARYSENSOR_MQTT
{attribute 'reflection' := ''}
FUNCTION_BLOCK FB_INPUT_BINARYSENSOR_MQTT EXTENDS FB_MQTT_BASE
VAR_INPUT
	BS: BOOL;
END_VAR
VAR_OUTPUT
	/// Follows the input but debounced 
	Q: BOOL;
	/// Event outputs only high for on clock cycle 
	EVENT: BOOL;
	EVENT_R: BOOL;
	EVENT_F: BOOL;
END_VAR
VAR
	/// object's full instance name 
	{attribute 'instance-path' := ''}
	{attribute 'noinit'}
	InstancePath: STRING;
	Startup: BOOL := TRUE;
	/// to debounce the physical input 
	FB_DEBOUNCE: OSCAT_BUILDING.DEBOUNCE;
	/// to detect a rising edge on the debounced signal 
	FB_R_TRIG: Standard.R_TRIG;
	/// to detect a falling edge on the debounced signal 
	FB_F_TRIG: Standard.F_TRIG;
	T_TurnOffDelay: TIME := TIME#0ms;
	FB_TurnOffDelayTimer: TOF;
	MqttDiscoveryMessage: MQTT_DISCOVERY_BINARY_SENSOR;
END_VAR

FB_DEBOUNCE(IN := BS,	
	TD := T#50MS, (* 2x cyle + 10ms *)
	PM := FALSE
	);
	
FB_TurnOffDelayTimer(IN:=FB_DEBOUNCE.Q,
	PT := T_TurnOffDelay,
	Q=>Q
	);

FB_R_TRIG(CLK := FB_TurnOffDelayTimer.Q);
FB_F_TRIG(CLK := FB_TurnOffDelayTimer.Q);

EVENT := FB_R_TRIG.Q OR FB_F_TRIG.Q;
EVENT_R := FB_R_TRIG.Q;
EVENT_F := FB_F_TRIG.Q;

IF (FB_R_TRIG.Q OR (Startup AND FB_DEBOUNCE.Q)) AND InitMqttDone THEN
	pMqttPublishQueue^.AddMessage(
		Payload := 'ON',
		Topic := CONCAT(MqttPublishTopicPrefix^, MqttPublishTopicSuffix),
		Qos := MQTT.QoS.ExactlyOnce,
		MqttRetain := TRUE
	);
	Startup:=FALSE;	
END_IF

IF (FB_F_TRIG.Q OR (Startup AND NOT(FB_DEBOUNCE.Q))) AND InitMqttDone THEN
	pMqttPublishQueue^.AddMessage(
		Payload := 'OFF',
		Topic := CONCAT(MqttPublishTopicPrefix^, MqttPublishTopicSuffix),
		Qos := MQTT.QoS.ExactlyOnce,
		MqttRetain := TRUE
	);
	Startup:=FALSE;	
END_IF

METHOD ConfigureFunctionBlock
VAR_INPUT
	T_TurnOffDelay: TIME;
END_VAR
THIS^.T_TurnOffDelay:=T_TurnOffDelay;
END_METHOD

METHOD InitMqtt
VAR_INPUT
	MQTTPublishPrefix: POINTER TO STRING;
	pMqttPublishQueue: POINTER TO FB_MqttPublishQueue;
END_VAR
SUPER^._InstancePath := THIS^.InstancePath; // Due to reflection its location is important

(*pass trough*)
THIS^.pMqttPublishQueue := pMqttPublishQueue;
THIS^.MqttPublishTopicPrefix:=MQTTPublishPrefix;
SUPER^.InitBaseMqtt();
END_METHOD

METHOD InitMqttDiscovery
VAR_INPUT
	Device: POINTER TO FB_PLC_MQTT_DISCOVERY_DEVICE;
	Name: STRING(255);
	DeviceClass: STRING(100) := 'smoke';
	overruleId: STRING(255) := '';
	meta: STRING(255) := '';
END_VAR
VAR
	id: STRING(255);
END_VAR
IF InitMqttDone AND NOT initMqttDiscoveryDone THEN
	
	IF CommonTypesAndFunctions.StrEquals(str1:= ADR(overruleId), str2:= ADR('')) THEN
		id := CONCAT(CONCAT(THIS^.DeviceName,'_'), THIS^.InstanceNamePt^); // 'FB_DI_PB_003'
	ELSE
		id := overruleId; // 'MY_PH_GND_HALL_01'
	END_IF
	
	Device^.CreateBinarySensorEntity(
		Id := id,
		Name := name,
		Meta := meta,
		StateTopic := THIS^.MQTTPublishTopic,
		PayloadOn := 'ON',
		PayloadOff := 'OFF',
		DeviceClass := DeviceClass);
		
	initMqttDiscoveryDone := TRUE;
END_IF
END_METHOD

END_FUNCTION_BLOCK

// FB_RS485_EASTRON_SDM_POWER_MQTT
{attribute 'reflection' := ''}
FUNCTION_BLOCK FB_RS485_EASTRON_SDM_POWER_MQTT IMPLEMENTS RS485Device
VAR_OUTPUT
	ACTIVEPOWER: REAL := 0;
	DataAvailable: BOOL := FALSE;
	Error: BOOL := FALSE;
END_VAR
VAR
	/// object's full instance name 
	{attribute 'noinit'}
	{attribute 'instance-path' := ''}
	InstanceName: STRING;
	Startup: BOOL := TRUE;
	InitMqttDone: BOOL;
	MqttPublishTopicPrefix: POINTER TO STRING;
	MqttPublishTopicSuffix: STRING(50);
	pMqttPublishQueue: POINTER TO FB_MqttPublishQueue;
	InitRS485Done: BOOL := FALSE;
	ActiveDevice: BOOL := FALSE;
	timerData: TON;
	isDataUpdated: BOOL := FALSE;
	DeviceType: RS485_EASTRON_SDM_Devices;
	SDM120AndSDM220RtuQuery: RS485_RtuQuery := (FunctionCode := 4, ReadAddress := 12, ReadQuantity := 2);
	SDM630RtuQuery: RS485_RtuQuery := (FunctionCode := 4, ReadAddress := 52, ReadQuantity := 2);
END_VAR

timerData();

IF isDataUpdated THEN
	isDataUpdated := FALSE;
	
	IF InitMqttDone THEN
		pMqttPublishQueue^.AddMessage(
			Payload := REAL_TO_STRING(ACTIVEPOWER),
			Topic := CONCAT(CONCAT(MqttPublishTopicPrefix^, MqttPublishTopicSuffix), '/ACTP' ),
			Qos := MQTT.QoS.ExactlyOnce,
			MqttRetain := FALSE
		);
	END_IF
END_IF

METHOD GetRtuQuery : RS485_RtuQuery
IF timerData.Q THEN
	THIS^.timerData.IN := FALSE;
	IF DeviceType = RS485_EASTRON_SDM_Devices.SDM120 OR  DeviceType = RS485_EASTRON_SDM_Devices.SDM220 THEN
		GetRtuQuery := THIS^.SDM120AndSDM220RtuQuery;		
	END_IF
	IF DeviceType = RS485_EASTRON_SDM_Devices.SDM630 THEN
		GetRtuQuery := THIS^.SDM630RtuQuery;		
	END_IF
END_IF
END_METHOD

METHOD InitMqtt
VAR_INPUT
	MQTTPublishPrefix: POINTER TO STRING;
	pMqttPublishQueue: POINTER TO FB_MqttPublishQueue;
END_VAR
VAR
	InstanceNamePt: POINTER TO STRING;
END_VAR
THIS^.pMqttPublishQueue := pMqttPublishQueue;
THIS^.MqttPublishTopicPrefix := MQTTPublishPrefix;

InstanceNamePt := CommonTypesAndFunctions.FindLastDot(ADR(THIS^.InstanceName)) + 1;
THIS^.MqttPublishTopicSuffix := InstanceNamePt^;

THIS^.InitMqttDone := TRUE;
END_METHOD

METHOD InitRS485
VAR_INPUT
	DataPollingInterval: TIME;
	DeviceAddress: BYTE;
	DeviceType: RS485_EASTRON_SDM_Devices;
END_VAR
THIS^.timerData.PT := DataPollingInterval;
THIS^.SDM120AndSDM220RtuQuery.DeviceId := DeviceAddress;
THIS^.SDM630RtuQuery.DeviceId := DeviceAddress;
THIS^.timerData.IN := TRUE;
THIS^.DeviceType := DeviceType;

THIS^.InitRS485Done := TRUE;
END_METHOD

METHOD ProcessDataArray
VAR_INPUT
	Error: POINTER TO BOOL;
	Data: POINTER TO ARRAY[0..124] OF WORD;
END_VAR
THIS^.Error := Error^;
THIS^.timerData.IN := TRUE;

IF Error^ THEN
	PubMqttMessage(Suffix := '/availability', Data := 'offline');
ELSE
	PubMqttMessage(Suffix := '/availability', Data := 'online');
END_IF

IF NOT Error^ THEN
	THIS^.ACTIVEPOWER := SwapWordsToReal(Data^[0], Data^[1]);
	THIS^.isDataUpdated := TRUE;
END_IF

ActiveDevice := FALSE;
END_METHOD

METHOD PubMqttMessage
VAR_INPUT
	Suffix: STRING(100);
	Data: STRING(100);
END_VAR
IF InitMqttDone THEN
		pMqttPublishQueue^.AddMessage(
			Payload := Data,
			Topic := CONCAT(CONCAT(MqttPublishTopicPrefix^, MqttPublishTopicSuffix), Suffix ),
			Qos := MQTT.QoS.ExactlyOnce,
			MqttRetain := FALSE
		);
END_IF
END_METHOD

METHOD RequestBusTime : BOOL
IF NOT InitRS485Done THEN	
	RequestBusTime := FALSE;	
ELSIF timerData.Q THEN
	RequestBusTime := TRUE;
ELSE
	RequestBusTime := FALSE;	
END_IF
END_METHOD

END_FUNCTION_BLOCK
